// TwinCAT 3 PLC project DAS_CoreSys
// ProgramVersion: 3.1.4024.0
// libraries:
//   AxisInterface_Type03, * (Beckhoff Automation)
//   BATW_Base, * (Beckhoff Automation)
//   Common Behaviour Model, * (3S - Smart Software Solutions GmbH)
//   Tc2_EtherCAT, * (Beckhoff Automation GmbH)
//   Tc2_Math, * (Beckhoff Automation GmbH)
//   Tc2_ModbusRTU, * (Beckhoff Automation GmbH)
//   Tc2_SerialCom, * (Beckhoff Automation GmbH)
//   Tc2_Standard, * (Beckhoff Automation GmbH)
//   Tc2_System, * (Beckhoff Automation GmbH)
//   Tc2_Utilities, * (Beckhoff Automation GmbH)
//   Tc3_JsonXml, * (Beckhoff Automation GmbH)
//   Tc3_MC2_AdvancedHoming, * (Beckhoff Automation GmbH)
//   Tc3_Module, * (Beckhoff Automation GmbH)
//   Tc3_PackML_V2, * (Beckhoff Automation GmbH)
//   Util, * (System)
// project tree:
//   / CoreSys.TcTTO, ModbusTask.TcTTO, MotionSync.TcTTO
//   Library/00_PackML/01_ObjectBase/ eModeChangeState.TcDUT, FB_ModeBase_V1.TcPOU, FB_ModeBase_V2.TcPOU, I_ErrorElement.TcIO, I_ErrorSubject.TcIO
//   Library/00_PackML/02_Mode/ E_Severity.TcDUT, E_UnitMode.TcDUT
//   Library/10_Machine/11_IOData/ GVL_EIP.TcGVL, GVL_Input.TcGVL, GVL_Output.TcGVL
//   Library/10_Machine/12_MachineControl/DUTs/ AxisNo.TcDUT, E_DataFrom.TcDUT, ST_ChangeIntoProduction.TcDUT, ST_CylinderMonitor.TcDUT, ST_MotorMonitor.TcDUT, ST_TableMoveCtrl.TcDUT, ST_TableMoveService.TcDUT, ST_TableMoveStatus.TcDUT, UnitNo.TcDUT
//   Library/10_Machine/12_MachineControl/DUTs/Cylinders/ ST_CylinderList.TcDUT, UNI_CylinderList.TcDUT
//   Library/10_Machine/12_MachineControl/DUTs/FanucRobot/ ST_FanucRobotList.TcDUT, UNI_FanucRobotList.TcDUT
//   Library/10_Machine/12_MachineControl/DUTs/Motor/ ST_MotorList.TcDUT, UNI_MotorList.TcDUT
//   Library/10_Machine/12_MachineControl/DUTs/Service/ ST_ServiceCtrl_Base.TcDUT, ST_ServiceStatus_Base.TcDUT
//   Library/10_Machine/12_MachineControl/DUTs/Setup/ E_ClipNo.TcDUT, ST_AllocateRobotCoordinate.TcDUT, ST_AllocateRobotPositionTable.TcDUT, ST_AxisPara.TcDUT, ST_AxisPara_Auto.TcDUT, ST_AxisPara_HalfAuto.TcDUT, ST_AxisPara_Homing.TcDUT, ST_AxisPara_Manual.TcDUT, ST_CylinderPara.TcDUT, ST_FanucRobotCCDSetting.TcDUT, ST_OutRobotCoordinate.TcDUT, ST_OutRobotPositionTable.TcDUT, ST_PositionTable.TcDUT, ST_SetupAxis.TcDUT, ST_SetupCylinder.TcDUT, ST_SetupFanucRobot.TcDUT, ST_SetupMotor.TcDUT, ST_SetupPara.TcDUT, ST_Setup_Light.TcDUT, ST_Setup_Mechanical.TcDUT
//   Library/10_Machine/12_MachineControl/ FB_MachineControl.TcPOU, GVL_Machine.TcGVL, GVL_Machine_Const.TcGVL
//   Library/10_Machine/12_MachineControl/Service/ FB_MachineHoming.TcPOU
//   Library/10_Machine/18_HMI_Handshake/DUTs/Allocated/ ST_Auto_Allocated.TcDUT, ST_AXIS_HOMING.TcDUT, ST_AXIS_JOG.TcDUT, ST_AXIS_PTP.TcDUT, ST_HalfAuto_Allocated.TcDUT, ST_HMI_ControlOutPut.TcDUT, ST_Manual_Allocated.TcDUT, ST_Manual_NeedleRobot.TcDUT, ST_Manual_Axis.TcDUT, ST_Manual_OutRobot.TcDUT, ST_Manual_PullOutCV.TcDUT, ST_Manual_Allocate.TcDUT, ST_Manual_TransCV.TcDUT, ST_Manual_TurnTable.TcDUT
//   Library/10_Machine/18_HMI_Handshake/DUTs/Component/ ST_DoubleValve.TcDUT, ST_MotorCommand.TcDUT, ST_SignleValve.TcDUT
//   Library/10_Machine/18_HMI_Handshake/DUTs/ E_AllocationJob.TcDUT
//   Library/10_Machine/18_HMI_Handshake/DUTs/IOMonitor/ ST_HMI_ControlInPut.TcDUT, ST_InputTables.TcDUT, ST_Input_IOMonitor.TcDUT, ST_Output_IOMonitor.TcDUT, ST_WheelhouseInput.TcDUT, ST_WheelhouseTour.TcDUT, ST_Wheelhouse_Layer.TcDUT, UNI_HMI_WheelHouseInput.TcDUT, UNI_HMI_WheelHouseInput2.TcDUT (excluded from build)
//   Library/10_Machine/18_HMI_Handshake/DUTs/Shipping/ ST_Auto_Shipping.TcDUT, ST_HalfAuto_Shipping.TcDUT, ST_HMI_ShippingArea.TcDUT, ST_Manual_Shipping.TcDUT
//   Library/10_Machine/18_HMI_Handshake/DUTs/Status/ ST_AllocateStatus.TcDUT, ST_Auto_Status.TcDUT, ST_AXES_STATUS.TcDUT, ST_MotorStatus.TcDUT, ST_SINGLEAXIS_STATUS.TcDUT, ST_CylinderStatus.TcDUT, ST_HalfAuto_Status.TcDUT, ST_HMI_MachineStatus.TcDUT, ST_Manual_Status.TcDUT, ST_ShippingStatus.TcDUT, ST_StorageStatus.TcDUT
//   Library/10_Machine/18_HMI_Handshake/DUTs/Storage/ ST_Auto_Storage.TcDUT, ST_HalfAuto_Storage.TcDUT, ST_HMI_ControlConvery.TcDUT, ST_Manual_FanucRobot.TcDUT, ST_Manual_Rack.TcDUT, ST_Manual_UpCV.TcDUT, ST_Manual_LowCV.TcDUT, ST_Manual_Storage.TcDUT
//   Library/10_Machine/18_HMI_Handshake/ FB_HmiHandShake.TcPOU, GVL_ADS.TcGVL, GVL_HMI.TcGVL
//   Library/10_Machine/18_HMI_Handshake/OLD_DUTs/DataCore/ E_BoxHookPoint.TcDUT, E_BufferArea.TcDUT, E_BoxStatus.TcDUT, E_LayerPoint.TcDUT, E_MachineMode.TcDUT, E_mode.TcDUT, E_NeedleClip.TcDUT, E_Location.TcDUT, E_MachineTask.TcDUT, E_NeedlePoint.TcDUT, E_OutRobotClip.TcDUT, E_OutRobotPoint.TcDUT, E_PlateHookPoint.TcDUT, st_AllocatingNeedleInfo.TcDUT, ST_AllocationJobBatchModeInfo.TcDUT, st_BoxHookStationMove.TcDUT, ST9_ChangeBox.TcDUT, st_ChangeBoxesData.TcDUT, ST0_ChangeBoxesInfo.TcDUT, ST1_ChangeBoxInfo.TcDUT, st_LayerStationMove.TcDUT, ST_Mode.TcDUT, ST_Output.TcDUT, ST_DischargeDataInfo.TcDUT, ST_Feeding.TcDUT, ST_FeedingDataFeeback.TcDUT, ST_FeedingDataInfo.TcDUT, ST_GetBox.TcDUT, st_NeedleAction.TcDUT, st_NeedleActionBatch.TcDUT, ST_NeedleAllocatefeeback.TcDUT, ST_NeedleAllocateinfo.TcDUT, ST_ChangeAllocate.TcDUT, ST_NeedleChangeAllocateInfo.TcDUT, ST_NeedleRemove.TcDUT, ST_NeedleRemoveAllocate.TcDUT, st_OutRobotMove.TcDUT, ST_PCTask.TcDUT, st_PlateHookStationMove.TcDUT, ST_PlateOrder.TcDUT, E_StationOrder.TcDUT, ST_ACTIVEDATA.TcDUT, ST_ActiveResult.TcDUT, ST_AllocationData.TcDUT, ST_AllocationInfo.TcDUT, ST_AllocationJobBatchMode_Reverse.TcDUT, st_ADSBaseParaCore.TcDUT, st_ADSMotoCore.TcDUT, st_ADSMotoMoveCore.TcDUT, st_AllocateParameterCore.TcDUT, st_RegionHome.TcDUT, ST_SheepingPicture.TcDUT, ST_SheepingPictureFeeback.TcDUT, ST_SheepingPictureInfo.TcDUT, ST_SixRobotAction.TcDUT, ST_SixRobotActionFeeback.TcDUT, ST_SixRobotActionInfo.TcDUT, st_SixRobotAreaMove.TcDUT, st_SixRobotPTP.TcDUT, ST_WarehouseBack.TcDUT, ST_WarehouseBackFeeback.TcDUT, ST_WarehouseBackInfo.TcDUT, ST_WarehouseGetBox.TcDUT, ST_ClampingToPlate.TcDUT, st_DASCalibrationData.TcDUT, ST_GetBoxData.TcDUT, ST_GetBoxInfo.TcDUT, ST_InformationExchange.TcDUT, ST_MachineAdjust.TcDUT, ST_MachineTask.TcDUT, ST_Needle.TcDUT, ST_NeedleChageBox.TcDUT, st_NeedleChageBoxData.TcDUT, ST_NeedleWarehouse.TcDUT, ST_NeedleWarehouseData.TcDUT, ST_SixRobotGetOrPut.TcDUT, st_WarehouseData.TcDUT
//   Library/10_Machine/18_HMI_Handshake/Service/DUTs/AllocateBatchMode/ st_AllocateMoveAutoBatchMode_Ctrl.TcDUT, st_AllocateMoveAutoBatchMode_Status.TcDUT, st_Coordinate.TcDUT, ST_Cylinders.TcDUT, st_RoundBeltAutoSingleMove_Ctrl.TcDUT, U_Cylinders.TcDUT
//   Library/10_Machine/18_HMI_Handshake/Service/DUTs/ ST_HMI_Handshake.TcDUT
//   Library/10_Machine/19_Device/EL1889/ ST_EbusDI16.TcDUT, ST_EbusInputModule.TcDUT, ST_InputTable.TcDUT, ST_InputTable_Mitsubishi.TcDUT, uni_InputModule.TcDUT
//   Library/10_Machine/19_Device/EL2889/ ST_EbusDO16.TcDUT, ST_EbusOutputModule.TcDUT, ST_OutputTable.TcDUT, ST_OutputTables.TcDUT, uni_OutputModule.TcDUT
//   Library/10_Machine/19_Device/FanucRobot/DUTs/ E_ClampAction.TcDUT, E_FanucRobotOpMode.TcDUT, E_PullOutConveyorPosition.TcDUT, E_RobotAddress.TcDUT, ST_AutoMode_ShippingRobot_MoveAbs.TcDUT, ST_CCD_ZoneUse.TcDUT, ST_FanucUI1.TcDUT, ST_FanucUO1.TcDUT, ST_Fanuc_AbsMove.TcDUT, ST_Fanuc_GeneralCommand.TcDUT, ST_Fanuc_GeneralCommand_1.TcDUT, ST_Fanuc_Status.TcDUT, ST_Fanuc_WarehouseHandshake.TcDUT, ST_IntToBool.TcDUT, ST_ReadWriteParaCmd.TcDUT, ST_ReadWriteParaStatus.TcDUT
//   Library/10_Machine/19_Device/FanucRobot/ FB_FanucRobot_Basic.TcPOU
//   Library/20_MachineUnits/21_StorageArea/210_Cabinet/DUTs/ E_CabinetJob.TcDUT, st_LayerStatus.TcDUT, st_WarehouseLayer.TcDUT, st_WarehouseList.TcDUT, U_Bits_To_stStatus.TcDUT, _st_LayerStatus.TcDUT, _st_WareHouseLayer.TcDUT, _st_WarehouseList.TcDUT
//   Library/20_MachineUnits/21_StorageArea/210_Cabinet/ FB_WareHouse.TcPOU
//   Library/20_MachineUnits/21_StorageArea/210_Cabinet/Services/ FB_FeedInBox.TcPOU, FB_ReloadBox.TcPOU
//   Library/20_MachineUnits/21_StorageArea/Duts/ E_CabinetJob.TcDUT (excluded from build), E_FeedInAction.TcDUT, E_ReloadRoundBoxAction.TcDUT, st_RobotAbsMove_Ctrl.TcDUT, st_RobotAbsMove_Status.TcDUT, st_RobotWarehouseMove_Ctrl.TcDUT, st_RobotWarehouseMove_Status.TcDUT, ST_StorageService.TcDUT
//   Library/20_MachineUnits/21_StorageArea/ FB_StorageArea.TcPOU
//   Library/20_MachineUnits/21_StorageArea/Service/ FB_AddBoxes_v2.TcPOU, FB_BoxSupplyCtrl.TcPOU, FB_DiameterMovement.TcPOU, FB_FeedInEmptyBoxWithRobot.TcPOU, FB_LowerFeedInConveyor.TcPOU, FB_ReloadRoundBeltBoxWithRobot.TcPOU, FB_RobotAbsMove.TcPOU, FB_RobotRegionMove_AllocatedConveyor.TcPOU, FB_RobotRegionMove_BufferArea.TcPOU, FB_RobotRegionMove_FeedInConveyor.TcPOU, FB_RobotRegionMove_PullOutConveyor.TcPOU, FB_RobotRegionMove_RoundBelt.TcPOU, FB_StorageHoming.TcPOU, FB_UpperFeedInConveyor.TcPOU, FB_WareHouseWithRobotMove.TcPOU
//   Library/20_MachineUnits/22_AllocateArea/Duts/Enums/ E_RoundBeltControlAccess.TcDUT
//   Library/20_MachineUnits/22_AllocateArea/Duts/ E_Pistons.TcDUT, F_Even.TcPOU, ST_AllocateService.TcDUT, ST_DuoCylinders.TcDUT, st_RoundBeltAutoSingleMove_Status.TcDUT, Uni_DuoCylinders.TcDUT
//   Library/20_MachineUnits/22_AllocateArea/ FB_AllocateAreaWithRoundbelt.TcPOU, FB_AllocateAreaWithXPlanar.TcPOU
//   Library/20_MachineUnits/22_AllocateArea/FUNs/ FUN_GetNeedleCoordinates.TcPOU, FUN_GetSyncGroup_AllocationJob.TcPOU
//   Library/20_MachineUnits/22_AllocateArea/Service/ FB_AllocateRobotNeedlingMove.TcPOU, FB_AllocateMoveAutoBatchMode.TcPOU, FB_AllocateMoveAutoBatchMode_Reverse.TcPOU, FB_OutRobot_EmptyBoxMove.TcPOU, FB_OutRobot_RareBoxMove.TcPOU, FB_OutRobot_BoxMoveReverse.TcPOU, FB_OutRobot_BoxMoveTurnTableToRoundBelt.TcPOU, FB_PullOutConveyorAction.TcPOU, FB_PullOutConveyorBtnCtrl.TcPOU, FB_RoundBeltService.TcPOU, FB_AllocateAreaHome.TcPOU, FB_SameSizeCVCamera.TcPOU, FB_DifferentCVCamera.TcPOU, FB_TurnTableService.TcPOU
//   Library/20_MachineUnits/23_ShippingArea/Duts/ ST_ShippingService.TcDUT
//   Library/20_MachineUnits/23_ShippingArea/ FB_ShippingArea.TcPOU
//   Library/20_MachineUnits/23_ShippingArea/Service/ FB_ShippingHoming.TcPOU, FB_ShippingRobot_TransmitCVEnd.TcPOU, FB_ShippingRobot_Left.TcPOU, FB_ShippingRobot_Right.TcPOU
//   Library/99_Utilities/Duts/ E_SignalTowerLampMode.TcDUT, ST_BoolList.TcDUT, ST_SignalTower.TcDUT, uni_IntToBool.TcDUT
//   Library/99_Utilities/ErrorHandling/ FB_ErrorHandler.TcPOU, FB_ErrorHandler_OLD.TcPOU (excluded from build), FB_ErrorHandler_abond.TcPOU (excluded from build), FB_ErrorHandling.TcPOU (excluded from build)
//   Library/99_Utilities/ FB_CylinderManualCtrl.TcPOU, FB_EdgeDetect.TcPOU, FB_MotorManualCtrl.TcPOU, FB_SignalGen.TcPOU, FB_SignalTower.TcPOU, FB_TableMove.TcPOU, FB_XY_Move.TcPOU, FB_XY_PickAndPlace.TcPOU, F_FtoPT.TcPOU
//   Library/99_Utilities/FUNCTION/ FUN_CheckAxisAllowMove.TcPOU, FUN_GetPositionTableData.TcPOU, FUN_MachineState.TcPOU, FUN_ResetStorageCylinder.TcPOU, FUN_RetractStorageCylinder.TcPOU
//   POUs/CheckProg/ CheckBounds.TcPOU, CheckDivDInt.TcPOU, CheckDivLInt.TcPOU, CheckDivLReal.TcPOU, CheckDivReal.TcPOU, CheckLRangeSigned.TcPOU, CheckLRangeUnsigned.TcPOU, CheckPointer.TcPOU, CheckRangeSigned.TcPOU, CheckRangeUnsigned.TcPOU
//   POUs/ DAS_CoreSys.TcPOU, DAS_MotionSync.TcPOU
//   POUs/ModbusRTU/00_BaseFBs/01_FB_ObjectBase/DUTs/ E_MethodStatus_Basic.TcDUT, ST_CmdContent.TcDUT, ST_MsgContent.TcDUT
//   POUs/ModbusRTU/00_BaseFBs/01_FB_ObjectBase/ FB_ObjectBase.TcPOU, FB_ObjectBase_V2.TcPOU
//   POUs/ModbusRTU/00_BaseFBs/01_FB_ObjectBase/GVLs/ Para_ObjectBase.TcGVL
//   POUs/ModbusRTU/00_BaseFBs/01_FB_ObjectBase/ITFs/ IBasicElement.TcIO
//   POUs/ModbusRTU/ ComModbusRTU.TcPOU
//   POUs/ModbusRTU/SerialComTask/DUTs/ un_RS485States.TcDUT, un_RS485States_all.TcDUT
//   POUs/ModbusRTU/SerialComTask/ FB_CommunicateModbusRTU.TcPOU
// real-time tasks:
//   TASK CoreSys: cycle T#10ms, priority 20, ADS port 350
//   TASK MotionSync: cycle T#2ms, priority 1, ADS port 351
//   TASK EIP_Task: cycle T#2ms, priority 2, ADS port 301
//   TASK ModbusTask: cycle T#5ms, priority 21, ADS port 352
// motion (NC):
//   TASK NC-Task 1 SAF: cycle T#2ms, priority 4, ADS port 501
//   TASK NC-Task 1 SVB: cycle T#2ms, priority 8, ADS port 511
//   AXIS Axis 1|TurnTable (id 1)
//     General: UnitName=°
//     Dynamic: Acceleration=1800, Deceleration=1800, Jerk=10800
//     Velo: SlowManual=6, FastManual=60, Maximum=600
//     OtherSettings: AllowMotionCmdToSlave=true
//     encoder EncType=19
//       EncPara: ScaleFactorNumerator=120, ScaleFactorDenominator=83886080, MaxCount=#xffffffff
//         SoftEndMaxControl: Range=350
//         Inc: RefSoftSyncMask=#x0000ffff
//     drive DrvType=16
//       DrvPara: MaxCount=#xffffffff, DriveControlDWord=#x00020100
//         Analog: VeloReferenz=600, TorqueSetpointScale=10, ScaleFactorActTorque=0.1
//         TimeComp: TaskDelayCycles=1
//     controller CtrType=1
//       CtrPara: PriorControlFactor=1
//         PosDiffControl: Enable=false
//         Observer: BandWidth=20
//   AXIS Axis 2|RoundBelt (id 2)
//     General: UnitFlags=#x00000004
//     Dynamic: AccelerationMaximum=3900, DecelerationMaximum=3900, Acceleration=3900, Deceleration=3900, Jerk=30000
//     Velo: SlowManual=6, FastManual=300, Maximum=500
//     OtherSettings: AllowMotionCmdToSlave=true
//     encoder EncType=19
//       EncPara: ScaleFactorNumerator=500, ScaleFactorDenominator=167772160, ModuloFactor=2800, MaxCount=#xffffffff
//         Inc: RefSoftSyncMask=#x0000ffff
//     drive DrvType=16
//       DrvPara: MaxCount=#xffffffff, DriveControlDWord=#x00020100
//         Analog: VeloReferenz=500, TorqueSetpointScale=10, ScaleFactorActTorque=0.1
//         TimeComp: TaskDelayCycles=1
//     controller CtrType=1
//       CtrPara: PriorControlFactor=1
//         PosDiffControl: Range=10
//         Observer: BandWidth=20
//   AXIS Axis 3|AllocateRobot_X (id 3)
//     Dynamic: Acceleration=12000, Deceleration=12000, Jerk=360000
//     Velo: SlowManual=6, FastManual=60, Maximum=800
//     OtherSettings: AllowMotionCmdToSlave=true
//     encoder EncType=19
//       EncPara: ScaleFactorNumerator=36, ScaleFactorDenominator=8388608, MaxCount=#xffffffff
//         Inc: RefSoftSyncMask=#x0000ffff
//     drive DrvType=16
//       DrvPara: MaxCount=#xffffffff, DriveControlDWord=#x00020100
//         Analog: TorqueSetpointScale=10, ScaleFactorActTorque=0.1
//         TimeComp: TaskDelayCycles=1
//     controller CtrType=1
//       CtrPara: PriorControlFactor=1
//         Observer: BandWidth=20
//   AXIS Axis 4|AllocateRobot_Y (id 4)
//     Dynamic: Acceleration=15000, Deceleration=15000, Jerk=225000
//     OtherSettings: AllowMotionCmdToSlave=true
//     encoder EncType=19
//       EncPara: ScaleFactorNumerator=16, ScaleFactorDenominator=8388608, Inverse=true, MaxCount=#xffffffff
//         Inc: RefSoftSyncMask=#x0000ffff
//     drive DrvType=16
//       DrvPara: Inverse=true, MaxCount=#xffffffff, DriveControlDWord=#x00020100
//         Analog: TorqueSetpointScale=10, ScaleFactorActTorque=0.1
//         TimeComp: TaskDelayCycles=1
//     controller CtrType=1
//       CtrPara: PriorControlFactor=1
//         PosDiffControl: Range=10
//         Observer: BandWidth=20
//   AXIS Axis 5|OutRobot_X (id 5)
//     Dynamic: Acceleration=11250, Deceleration=11250, Jerk=168750
//     Velo: SlowManual=6, FastManual=60, Maximum=1500
//     OtherSettings: AllowMotionCmdToSlave=true
//     encoder EncType=19
//       EncPara: ScaleFactorNumerator=30, ScaleFactorDenominator=8388608, MaxCount=#xffffffff
//     drive DrvType=16
//       DrvPara: MaxCount=#xffffffff, DriveControlDWord=#x00020100
//         Analog: TorqueSetpointScale=10, ScaleFactorActTorque=0.1
//         TimeComp: TaskDelayCycles=1
//     controller CtrType=1
//       CtrPara: PriorControlFactor=1
//         PosDiffControl: Range=10
//         Observer: BandWidth=20
//   AXIS Axis 6|OutRobot_Y (id 6)
//     Dynamic: Acceleration=6000, Deceleration=6000, Jerk=36000
//     Velo: SlowManual=6, FastManual=60
//     OtherSettings: AllowMotionCmdToSlave=true
//     encoder EncType=19
//       EncPara: ScaleFactorNumerator=40, ScaleFactorDenominator=8388608, MaxCount=#xffffffff
//     drive DrvType=16
//       DrvPara: MaxCount=#xffffffff, DriveControlDWord=#x00020100
//         Analog: TorqueSetpointScale=10, ScaleFactorActTorque=0.1
//         TimeComp: TaskDelayCycles=1
//     controller CtrType=1
//       CtrPara: PriorControlFactor=1
//         PosDiffControl: Range=10
//         Observer: BandWidth=20
//   AXIS Axis 7|RackMotor (id 7)
//     Dynamic: Acceleration=800.624, Deceleration=800.624, Jerk=1167.58
//     Velo: SlowManual=5, FastManual=100, Maximum=732
//     OtherSettings: AllowMotionCmdToSlave=true
//     encoder EncType=4
//       EncPara: ScaleFactorNumerator=90, ScaleFactorDenominator=980, MaxCount=#xffffffff
//     drive DrvType=23
//       Analog: VeloReferenz=732, TorqueSetpointScale=10, ScaleFactorActTorque=0.1
//       TimeComp: TaskDelayCycles=1
//     controller CtrType=1
//       CtrPara: PriorControlFactor=1
//         PosDiffControl: Enable=false
//         PID: PosKp=90
//         Observer: BandWidth=20
// I/O:
//   DEVICE Device 1 (EtherCAT) Storage, AmsNetId 169.254.53.69.2.1
//     Term 1 (EK1200) [EK1200-5000 EtherCAT Power supply (2A E-Bus)]
//       Term 2 (EL6021) [EL6021 Interface (RS422/485)]
//       Term 3 (EL6021) [EL6021 Interface (RS422/485)]
//       Term 4 (EL6021) [EL6021 Interface (RS422/485)]
//       Term 5 (EL6021) [EL6021 Interface (RS422/485)]
//       Term 6 (EL1889)_01(X6) [EL1889 16Ch. Dig. Input 24V, 3ms, negative]
//       Term 7 (EL1889)_02(X7) [EL1889 16Ch. Dig. Input 24V, 3ms, negative]
//       Term 8 (EL1889)_03(X9) [EL1889 16Ch. Dig. Input 24V, 3ms, negative]
//       Term 9 (EL1889)_04(X10) [EL1889 16Ch. Dig. Input 24V, 3ms, negative]
//       Term 10 (EL2889)_01(Y4) [EL2889 16Ch. Dig. Output 24V, 0.5A, negative]
//       Term 11 (EL2889)_02(Y5) [EL2889 16Ch. Dig. Output 24V, 0.5A, negative]
//       Term 12 (EL2889)_03(Y6) [EL2889 16Ch. Dig. Output 24V, 0.5A, negative]
//       Term 13 (EL2889)_04(Y7) [EL2889 16Ch. Dig. Output 24V, 0.5A, negative]
//       Term 14 (EL2889)_05(Y8) [EL2889 16Ch. Dig. Output 24V, 0.5A, negative]
//       Term 59 (EL9410) [EL9410 E-Bus Power Supplier  (Diagnostics)]
//       Term 15 (EL2889)_06(Y10) [EL2889 16Ch. Dig. Output 24V, 0.5A, negative]
//       Term 17 (EL2889)_07(Y11) [EL2889 16Ch. Dig. Output 24V, 0.5A, negative]
//       Term 18 (EL7342) [EL7342 2Ch. DC motor output stage (50V, 3.5A)]
//       Term 19 (EL6652) [EL6652 EtherNet/IP Scanner (Master)]
//       Term 20 (EL9011) [EL9011 End Terminal]
//   DEVICE Device 4 (EtherCAT) Allocate, AmsNetId 169.254.53.69.5.1
//     Box 21 (CU2508) [CU2508 Ethernet Port]
//     Term 22 (EK1100) [EK1100 EtherCAT Coupler (2A E-Bus)]
//       Term 23 (EL1889)_05(X0) [EL1889 16Ch. Dig. Input 24V, 3ms, negative]
//       Term 24 (EL1889)_06(X1) [EL1889 16Ch. Dig. Input 24V, 3ms, negative]
//       Term 25 (EL1889)_07(X2) [EL1889 16Ch. Dig. Input 24V, 3ms, negative]
//       Term 26 (EL1889)_08(X3) [EL1889 16Ch. Dig. Input 24V, 3ms, negative]
//       Term 27 (EL1889)_09(X8) [EL1889 16Ch. Dig. Input 24V, 3ms, negative]
//       Term 28 (EL1889)_10(X11) [EL1889 16Ch. Dig. Input 24V, 3ms, negative]
//       Term 29 (EL2889)_08(Y0) [EL2889 16Ch. Dig. Output 24V, 0.5A, negative]
//       Term 30 (EL2889)_09(Y1) [EL2889 16Ch. Dig. Output 24V, 0.5A, negative]
//       Term 31 (EL2889)_10(Y2) [EL2889 16Ch. Dig. Output 24V, 0.5A, negative]
//       Term 32 (EL9410) [EL9410 E-Bus Power Supplier  (Diagnostics)]
//       Term 33 (EL1889)_11(X4) [EL1889 16Ch. Dig. Input 24V, 3ms, negative]
//       Term 15 (EL6652) [EL6652 EtherNet/IP Scanner (Master)]
//       Term 16 (EL9011) [EL9011 End Terminal]
//   DEVICE Device 5 (EtherCAT), AmsNetId 169.254.53.69.6.1
//     Box 37 (CU2508) [CU2508 Ethernet Port]
//     Drive 38 (MBDLT25BF) [MBDLT25BF]
//     Drive 39 (MCDLT35BF) [MCDLT35BF]
//     Drive 40 (MBDLT25BF) [MBDLT25BF]
//     Drive 41 (MADLT15BF) [MADLT15BF]
//     Drive 42 (MADLT15BF) [MADLT15BF]
//     Drive 43 (MBDLT25BF) [MBDLT25BF]
//   DEVICE Storage Fanuc Robot (ECAT EIP Scanner (EL6652)), AmsNetId 169.254.53.69.4.1
//     FANUC Robot R30iB+ // <INFO> 192.168.0.3, FANUC Robot R30iB+ (ProdCode: 4, Rev: 3.01, Mac: 00:e0:e4:c5:29:bd) </INFO> <EDS> C:\TwinCAT\3.1\Config\Io\EtherNetIP\FANUCROBOT0301_R30IBP.EDS </EDS>
//   DEVICE Device 6 (ECAT EIP Scanner (EL6652)), AmsNetId 169.254.53.69.7.1
//     FANUC Robot R30iB+ // <INFO> 192.168.0.13, FANUC Robot R30iB+ (ProdCode: 4, Rev: 3.01, Mac: 00:e0:e4:99:c3:31) </INFO> <EDS> C:\TwinCAT\3.1\Config\Io\EtherNetIP\FANUCROBOT0301_R30IBP.EDS </EDS>
//   DEVICE X001 (RT-Ethernet Adapter)
// variable links:
//   NC-Task 1 SAF/Axes/Axis 1|TurnTable <-> Device 5 (EtherCAT)/Drive 38 (MBDLT25BF)
//     Drive/Inputs/In/nDataIn1 <-> Transmit PDO mapping 1/Following error actual value
//     Drive/Inputs/In/nDcOutputTime <-> InfoData/DcOutputShift
//     Drive/Inputs/In/nState1 <-> Transmit PDO mapping 1/Statusword
//     Drive/Inputs/In/nState2 <-> Transmit PDO mapping 1/Statusword @bit 8
//     Drive/Inputs/In/nState4 @bit 1 <-> WcState/InputToggle
//     Drive/Inputs/In/nState4 <-> WcState/WcState
//     Drive/Inputs/In/nState5 <-> Transmit PDO mapping 1/Modes of operation display
//     Drive/Outputs/Out/nCtrl1 <-> Receive PDO mapping 1/Controlword
//     Drive/Outputs/Out/nCtrl2 <-> Receive PDO mapping 1/Controlword @bit 8
//     Drive/Outputs/Out/nCtrl5 <-> Receive PDO mapping 1/Modes of operation
//     Drive/Outputs/Out/nDataOut1 <-> Receive PDO mapping 1/Target position
//     Enc/Inputs/In/nDataIn1 <-> Transmit PDO mapping 1/Position actual value
//     Enc/Inputs/In/nDataIn3 <-> Transmit PDO mapping 1/Touch probe pos1 pos value
//     Enc/Inputs/In/nDcInputTime <-> InfoData/DcInputShift
//     Enc/Inputs/In/nState4 @bit 1 <-> WcState/InputToggle
//     Enc/Inputs/In/nState4 <-> WcState/WcState
//     Enc/Inputs/In/nState5 <-> Transmit PDO mapping 1/Touch probe status
//     Enc/Inputs/In/nState6 <-> Transmit PDO mapping 1/Touch probe status @bit 8
//     Enc/Outputs/Out/nCtrl5 <-> Receive PDO mapping 1/Touch probe function
//     Enc/Outputs/Out/nCtrl6 <-> Receive PDO mapping 1/Touch probe function @bit 8
//   NC-Task 1 SAF/Axes/Axis 2|RoundBelt <-> Device 5 (EtherCAT)/Drive 39 (MCDLT35BF)
//     Drive/Inputs/In/nDataIn1 <-> Transmit PDO mapping 1/Following error actual value
//     Drive/Inputs/In/nDataIn3[0] <-> Transmit PDO mapping 1/Torque actual value
//     Drive/Inputs/In/nDcOutputTime <-> InfoData/DcOutputShift
//     Drive/Inputs/In/nState1 <-> Transmit PDO mapping 1/Statusword
//     Drive/Inputs/In/nState2 <-> Transmit PDO mapping 1/Statusword @bit 8
//     Drive/Inputs/In/nState4 @bit 1 <-> WcState/InputToggle
//     Drive/Inputs/In/nState4 <-> WcState/WcState
//     Drive/Inputs/In/nState5 <-> Transmit PDO mapping 1/Modes of operation display
//     Drive/Outputs/Out/nCtrl1 <-> Receive PDO mapping 1/Controlword
//     Drive/Outputs/Out/nCtrl2 <-> Receive PDO mapping 1/Controlword @bit 8
//     Drive/Outputs/Out/nCtrl5 <-> Receive PDO mapping 1/Modes of operation
//     Drive/Outputs/Out/nDataOut1 <-> Receive PDO mapping 1/Target position
//     Enc/Inputs/In/nDataIn1 <-> Transmit PDO mapping 1/Position actual value
//     Enc/Inputs/In/nDataIn3 <-> Transmit PDO mapping 1/Touch probe pos1 pos value
//     Enc/Inputs/In/nDcInputTime <-> InfoData/DcInputShift
//     Enc/Inputs/In/nState4 @bit 1 <-> WcState/InputToggle
//     Enc/Inputs/In/nState4 <-> WcState/WcState
//     Enc/Inputs/In/nState5 <-> Transmit PDO mapping 1/Touch probe status
//     Enc/Inputs/In/nState6 <-> Transmit PDO mapping 1/Touch probe status @bit 8
//     Enc/Outputs/Out/nCtrl5 <-> Receive PDO mapping 1/Touch probe function
//     Enc/Outputs/Out/nCtrl6 <-> Receive PDO mapping 1/Touch probe function @bit 8
//   NC-Task 1 SAF/Axes/Axis 3|AllocateRobot_X <-> Device 5 (EtherCAT)/Drive 40 (MBDLT25BF)
//     Drive/Inputs/In/nDataIn1 <-> Transmit PDO mapping 1/Following error actual value
//     Drive/Inputs/In/nDcOutputTime <-> InfoData/DcOutputShift
//     Drive/Inputs/In/nState1 <-> Transmit PDO mapping 1/Statusword
//     Drive/Inputs/In/nState2 <-> Transmit PDO mapping 1/Statusword @bit 8
//     Drive/Inputs/In/nState4 @bit 1 <-> WcState/InputToggle
//     Drive/Inputs/In/nState4 <-> WcState/WcState
//     Drive/Inputs/In/nState5 <-> Transmit PDO mapping 1/Modes of operation display
//     Drive/Outputs/Out/nCtrl1 <-> Receive PDO mapping 1/Controlword
//     Drive/Outputs/Out/nCtrl2 <-> Receive PDO mapping 1/Controlword @bit 8
//     Drive/Outputs/Out/nCtrl5 <-> Receive PDO mapping 1/Modes of operation
//     Drive/Outputs/Out/nDataOut1 <-> Receive PDO mapping 1/Target position
//     Enc/Inputs/In/nDataIn1 <-> Transmit PDO mapping 1/Position actual value
//     Enc/Inputs/In/nDataIn3 <-> Transmit PDO mapping 1/Touch probe pos1 pos value
//     Enc/Inputs/In/nDcInputTime <-> InfoData/DcInputShift
//     Enc/Inputs/In/nState4 @bit 1 <-> WcState/InputToggle
//     Enc/Inputs/In/nState4 <-> WcState/WcState
//     Enc/Inputs/In/nState5 <-> Transmit PDO mapping 1/Touch probe status
//     Enc/Inputs/In/nState6 <-> Transmit PDO mapping 1/Touch probe status @bit 8
//     Enc/Outputs/Out/nCtrl5 <-> Receive PDO mapping 1/Touch probe function
//     Enc/Outputs/Out/nCtrl6 <-> Receive PDO mapping 1/Touch probe function @bit 8
//   NC-Task 1 SAF/Axes/Axis 4|AllocateRobot_Y <-> Device 5 (EtherCAT)/Drive 41 (MADLT15BF)
//     Drive/Inputs/In/nDataIn1 <-> Transmit PDO mapping 1/Following error actual value
//     Drive/Inputs/In/nDcOutputTime <-> InfoData/DcOutputShift
//     Drive/Inputs/In/nState1 <-> Transmit PDO mapping 1/Statusword
//     Drive/Inputs/In/nState2 <-> Transmit PDO mapping 1/Statusword @bit 8
//     Drive/Inputs/In/nState4 @bit 1 <-> WcState/InputToggle
//     Drive/Inputs/In/nState4 <-> WcState/WcState
//     Drive/Inputs/In/nState5 <-> Transmit PDO mapping 1/Modes of operation display
//     Drive/Outputs/Out/nCtrl1 <-> Receive PDO mapping 1/Controlword
//     Drive/Outputs/Out/nCtrl2 <-> Receive PDO mapping 1/Controlword @bit 8
//     Drive/Outputs/Out/nCtrl5 <-> Receive PDO mapping 1/Modes of operation
//     Drive/Outputs/Out/nDataOut1 <-> Receive PDO mapping 1/Target position
//     Enc/Inputs/In/nDataIn1 <-> Transmit PDO mapping 1/Position actual value
//     Enc/Inputs/In/nDataIn3 <-> Transmit PDO mapping 1/Touch probe pos1 pos value
//     Enc/Inputs/In/nDcInputTime <-> InfoData/DcInputShift
//     Enc/Inputs/In/nState4 @bit 1 <-> WcState/InputToggle
//     Enc/Inputs/In/nState4 <-> WcState/WcState
//     Enc/Inputs/In/nState5 <-> Transmit PDO mapping 1/Touch probe status
//     Enc/Inputs/In/nState6 <-> Transmit PDO mapping 1/Touch probe status @bit 8
//     Enc/Outputs/Out/nCtrl5 <-> Receive PDO mapping 1/Touch probe function
//     Enc/Outputs/Out/nCtrl6 <-> Receive PDO mapping 1/Touch probe function @bit 8
//   NC-Task 1 SAF/Axes/Axis 5|OutRobot_X <-> Device 5 (EtherCAT)/Drive 42 (MADLT15BF)
//     Drive/Inputs/In/nDataIn1 <-> Transmit PDO mapping 1/Following error actual value
//     Drive/Inputs/In/nDcOutputTime <-> InfoData/DcOutputShift
//     Drive/Inputs/In/nState1 <-> Transmit PDO mapping 1/Statusword
//     Drive/Inputs/In/nState2 <-> Transmit PDO mapping 1/Statusword @bit 8
//     Drive/Inputs/In/nState4 @bit 1 <-> WcState/InputToggle
//     Drive/Inputs/In/nState4 <-> WcState/WcState
//     Drive/Inputs/In/nState5 <-> Transmit PDO mapping 1/Modes of operation display
//     Drive/Outputs/Out/nCtrl1 <-> Receive PDO mapping 1/Controlword
//     Drive/Outputs/Out/nCtrl2 <-> Receive PDO mapping 1/Controlword @bit 8
//     Drive/Outputs/Out/nCtrl5 <-> Receive PDO mapping 1/Modes of operation
//     Drive/Outputs/Out/nDataOut1 <-> Receive PDO mapping 1/Target position
//     Enc/Inputs/In/nDataIn1 <-> Transmit PDO mapping 1/Position actual value
//     Enc/Inputs/In/nDataIn3 <-> Transmit PDO mapping 1/Touch probe pos1 pos value
//     Enc/Inputs/In/nDcInputTime <-> InfoData/DcInputShift
//     Enc/Inputs/In/nState4 @bit 1 <-> WcState/InputToggle
//     Enc/Inputs/In/nState4 <-> WcState/WcState
//     Enc/Inputs/In/nState5 <-> Transmit PDO mapping 1/Touch probe status
//     Enc/Inputs/In/nState6 <-> Transmit PDO mapping 1/Touch probe status @bit 8
//     Enc/Outputs/Out/nCtrl5 <-> Receive PDO mapping 1/Touch probe function
//     Enc/Outputs/Out/nCtrl6 <-> Receive PDO mapping 1/Touch probe function @bit 8
//   NC-Task 1 SAF/Axes/Axis 6|OutRobot_Y <-> Device 5 (EtherCAT)/Drive 43 (MBDLT25BF)
//     Drive/Inputs/In/nDataIn1 <-> Transmit PDO mapping 1/Following error actual value
//     Drive/Inputs/In/nDcOutputTime <-> InfoData/DcOutputShift
//     Drive/Inputs/In/nState1 <-> Transmit PDO mapping 1/Statusword
//     Drive/Inputs/In/nState2 <-> Transmit PDO mapping 1/Statusword @bit 8
//     Drive/Inputs/In/nState4 @bit 1 <-> WcState/InputToggle
//     Drive/Inputs/In/nState4 <-> WcState/WcState
//     Drive/Inputs/In/nState5 <-> Transmit PDO mapping 1/Modes of operation display
//     Drive/Outputs/Out/nCtrl1 <-> Receive PDO mapping 1/Controlword
//     Drive/Outputs/Out/nCtrl2 <-> Receive PDO mapping 1/Controlword @bit 8
//     Drive/Outputs/Out/nCtrl5 <-> Receive PDO mapping 1/Modes of operation
//     Drive/Outputs/Out/nDataOut1 <-> Receive PDO mapping 1/Target position
//     Enc/Inputs/In/nDataIn1 <-> Transmit PDO mapping 1/Position actual value
//     Enc/Inputs/In/nDataIn3 <-> Transmit PDO mapping 1/Touch probe pos1 pos value
//     Enc/Inputs/In/nDcInputTime <-> InfoData/DcInputShift
//     Enc/Inputs/In/nState4 @bit 1 <-> WcState/InputToggle
//     Enc/Inputs/In/nState4 <-> WcState/WcState
//     Enc/Inputs/In/nState5 <-> Transmit PDO mapping 1/Touch probe status
//     Enc/Inputs/In/nState6 <-> Transmit PDO mapping 1/Touch probe status @bit 8
//     Enc/Outputs/Out/nCtrl5 <-> Receive PDO mapping 1/Touch probe function
//     Enc/Outputs/Out/nCtrl6 <-> Receive PDO mapping 1/Touch probe function @bit 8
//   NC-Task 1 SAF/Axes/Axis 7|RackMotor <-> Device 1 (EtherCAT) Storage/Term 1 (EK1200)/Term 18 (EL7342)
//     Drive/Inputs/In/nState1 @bit 3 <-> DCM Status Channel 1/Status/Error
//     Drive/Inputs/In/nState1 @bit 5 <-> DCM Status Channel 1/Status/Moving negative
//     Drive/Inputs/In/nState1 @bit 4 <-> DCM Status Channel 1/Status/Moving positive
//     Drive/Inputs/In/nState1 @bit 1 <-> DCM Status Channel 1/Status/Ready
//     Drive/Inputs/In/nState1 <-> DCM Status Channel 1/Status/Ready to enable
//     Drive/Inputs/In/nState1 @bit 6 <-> DCM Status Channel 1/Status/Torque reduced
//     Drive/Inputs/In/nState1 @bit 2 <-> DCM Status Channel 1/Status/Warning
//     Drive/Inputs/In/nState2 @bit 3 <-> DCM Status Channel 1/Status/Digital input 1
//     Drive/Inputs/In/nState2 @bit 4 <-> DCM Status Channel 1/Status/Digital input 2
//     Drive/Inputs/In/nState2 @bit 5 <-> DCM Status Channel 1/Status/Sync error
//     Drive/Inputs/In/nState2 @bit 7 <-> DCM Status Channel 1/Status/TxPDO Toggle
//     Drive/Inputs/In/nState4 @bit 1 <-> WcState/InputToggle
//     Drive/Inputs/In/nState4 <-> WcState/WcState
//     Drive/Outputs/Out/nCtrl1 <-> DCM Control Channel 1/Control/Enable
//     Drive/Outputs/Out/nCtrl1 @bit 2 <-> DCM Control Channel 1/Control/Reduce torque
//     Drive/Outputs/Out/nCtrl1 @bit 1 <-> DCM Control Channel 1/Control/Reset
//     Drive/Outputs/Out/nCtrl1 @bit 3 <-> DCM Control Channel 1/Control/Threshold active
//     Drive/Outputs/Out/nDataOut2[0] <-> DCM Velocity Channel 1/Velocity
//     Enc/Inputs/In/nDataIn1 <-> ENC Status Channel 1/Counter value
//     Enc/Inputs/In/nDataIn2 <-> ENC Status Channel 1/Latch value
//     Enc/Inputs/In/nState1 @bit 4 <-> ENC Status Channel 1/Status/Counter overflow
//     Enc/Inputs/In/nState1 @bit 3 <-> ENC Status Channel 1/Status/Counter underflow
//     Enc/Inputs/In/nState1 @bit 7 <-> ENC Status Channel 1/Status/Extrapolation stall
//     Enc/Inputs/In/nState1 @bit 1 <-> ENC Status Channel 1/Status/Latch extern valid
//     Enc/Inputs/In/nState1 @bit 2 <-> ENC Status Channel 1/Status/Set counter done
//     Enc/Inputs/In/nState2 @bit 4 <-> ENC Status Channel 1/Status/Status of extern latch
//     Enc/Inputs/In/nState2 <-> ENC Status Channel 1/Status/Status of input A
//     Enc/Inputs/In/nState2 @bit 1 <-> ENC Status Channel 1/Status/Status of input B
//     Enc/Inputs/In/nState2 @bit 5 <-> ENC Status Channel 1/Status/Sync error
//     Enc/Inputs/In/nState2 @bit 7 <-> ENC Status Channel 1/Status/TxPDO Toggle
//     Enc/Inputs/In/nState4 @bit 1 <-> WcState/InputToggle
//     Enc/Inputs/In/nState4 <-> WcState/WcState
//     Enc/Outputs/Out/nCtrl1 @bit 3 <-> ENC Control Channel 1/Control/Enable latch extern on negative edge
//     Enc/Outputs/Out/nCtrl1 @bit 1 <-> ENC Control Channel 1/Control/Enable latch extern on positive edge
//     Enc/Outputs/Out/nCtrl1 @bit 2 <-> ENC Control Channel 1/Control/Set counter
//     Enc/Outputs/Out/nDataOut1 <-> ENC Control Channel 1/Set counter value
//   DAS_CoreSys/DAS_CoreSys Instance <-> Device 1 (EtherCAT) Storage/Term 1 (EK1200)/Term 10 (EL2889)_01(Y4)
//     ModbusTask Outputs/GVL_Output.uniDO.stEbusDO.EL2889_01.DO1 <-> Channel 1/Output
//     ModbusTask Outputs/GVL_Output.uniDO.stEbusDO.EL2889_01.DO10 <-> Channel 10/Output
//     ModbusTask Outputs/GVL_Output.uniDO.stEbusDO.EL2889_01.DO11 <-> Channel 11/Output
//     ModbusTask Outputs/GVL_Output.uniDO.stEbusDO.EL2889_01.DO12 <-> Channel 12/Output
//     ModbusTask Outputs/GVL_Output.uniDO.stEbusDO.EL2889_01.DO13 <-> Channel 13/Output
//     ModbusTask Outputs/GVL_Output.uniDO.stEbusDO.EL2889_01.DO14 <-> Channel 14/Output
//     ModbusTask Outputs/GVL_Output.uniDO.stEbusDO.EL2889_01.DO15 <-> Channel 15/Output
//     ModbusTask Outputs/GVL_Output.uniDO.stEbusDO.EL2889_01.DO16 <-> Channel 16/Output
//     ModbusTask Outputs/GVL_Output.uniDO.stEbusDO.EL2889_01.DO2 <-> Channel 2/Output
//     ModbusTask Outputs/GVL_Output.uniDO.stEbusDO.EL2889_01.DO3 <-> Channel 3/Output
//     ModbusTask Outputs/GVL_Output.uniDO.stEbusDO.EL2889_01.DO4 <-> Channel 4/Output
//     ModbusTask Outputs/GVL_Output.uniDO.stEbusDO.EL2889_01.DO5 <-> Channel 5/Output
//     ModbusTask Outputs/GVL_Output.uniDO.stEbusDO.EL2889_01.DO6 <-> Channel 6/Output
//     ModbusTask Outputs/GVL_Output.uniDO.stEbusDO.EL2889_01.DO7 <-> Channel 7/Output
//     ModbusTask Outputs/GVL_Output.uniDO.stEbusDO.EL2889_01.DO8 <-> Channel 8/Output
//     ModbusTask Outputs/GVL_Output.uniDO.stEbusDO.EL2889_01.DO9 <-> Channel 9/Output
//   DAS_CoreSys/DAS_CoreSys Instance <-> Device 1 (EtherCAT) Storage/Term 1 (EK1200)/Term 11 (EL2889)_02(Y5)
//     ModbusTask Outputs/GVL_Output.uniDO.stEbusDO.EL2889_02.DO1 <-> Channel 1/Output
//     ModbusTask Outputs/GVL_Output.uniDO.stEbusDO.EL2889_02.DO10 <-> Channel 10/Output
//     ModbusTask Outputs/GVL_Output.uniDO.stEbusDO.EL2889_02.DO11 <-> Channel 11/Output
//     ModbusTask Outputs/GVL_Output.uniDO.stEbusDO.EL2889_02.DO12 <-> Channel 12/Output
//     ModbusTask Outputs/GVL_Output.uniDO.stEbusDO.EL2889_02.DO13 <-> Channel 13/Output
//     ModbusTask Outputs/GVL_Output.uniDO.stEbusDO.EL2889_02.DO14 <-> Channel 14/Output
//     ModbusTask Outputs/GVL_Output.uniDO.stEbusDO.EL2889_02.DO15 <-> Channel 15/Output
//     ModbusTask Outputs/GVL_Output.uniDO.stEbusDO.EL2889_02.DO16 <-> Channel 16/Output
//     ModbusTask Outputs/GVL_Output.uniDO.stEbusDO.EL2889_02.DO2 <-> Channel 2/Output
//     ModbusTask Outputs/GVL_Output.uniDO.stEbusDO.EL2889_02.DO3 <-> Channel 3/Output
//     ModbusTask Outputs/GVL_Output.uniDO.stEbusDO.EL2889_02.DO4 <-> Channel 4/Output
//     ModbusTask Outputs/GVL_Output.uniDO.stEbusDO.EL2889_02.DO5 <-> Channel 5/Output
//     ModbusTask Outputs/GVL_Output.uniDO.stEbusDO.EL2889_02.DO6 <-> Channel 6/Output
//     ModbusTask Outputs/GVL_Output.uniDO.stEbusDO.EL2889_02.DO7 <-> Channel 7/Output
//     ModbusTask Outputs/GVL_Output.uniDO.stEbusDO.EL2889_02.DO8 <-> Channel 8/Output
//     ModbusTask Outputs/GVL_Output.uniDO.stEbusDO.EL2889_02.DO9 <-> Channel 9/Output
//   DAS_CoreSys/DAS_CoreSys Instance <-> Device 1 (EtherCAT) Storage/Term 1 (EK1200)/Term 12 (EL2889)_03(Y6)
//     ModbusTask Outputs/GVL_Output.uniDO.stEbusDO.EL2889_03.DO1 <-> Channel 1/Output
//     ModbusTask Outputs/GVL_Output.uniDO.stEbusDO.EL2889_03.DO10 <-> Channel 10/Output
//     ModbusTask Outputs/GVL_Output.uniDO.stEbusDO.EL2889_03.DO11 <-> Channel 11/Output
//     ModbusTask Outputs/GVL_Output.uniDO.stEbusDO.EL2889_03.DO12 <-> Channel 12/Output
//     ModbusTask Outputs/GVL_Output.uniDO.stEbusDO.EL2889_03.DO13 <-> Channel 13/Output
//     ModbusTask Outputs/GVL_Output.uniDO.stEbusDO.EL2889_03.DO14 <-> Channel 14/Output
//     ModbusTask Outputs/GVL_Output.uniDO.stEbusDO.EL2889_03.DO15 <-> Channel 15/Output
//     ModbusTask Outputs/GVL_Output.uniDO.stEbusDO.EL2889_03.DO16 <-> Channel 16/Output
//     ModbusTask Outputs/GVL_Output.uniDO.stEbusDO.EL2889_03.DO2 <-> Channel 2/Output
//     ModbusTask Outputs/GVL_Output.uniDO.stEbusDO.EL2889_03.DO3 <-> Channel 3/Output
//     ModbusTask Outputs/GVL_Output.uniDO.stEbusDO.EL2889_03.DO4 <-> Channel 4/Output
//     ModbusTask Outputs/GVL_Output.uniDO.stEbusDO.EL2889_03.DO5 <-> Channel 5/Output
//     ModbusTask Outputs/GVL_Output.uniDO.stEbusDO.EL2889_03.DO6 <-> Channel 6/Output
//     ModbusTask Outputs/GVL_Output.uniDO.stEbusDO.EL2889_03.DO7 <-> Channel 7/Output
//     ModbusTask Outputs/GVL_Output.uniDO.stEbusDO.EL2889_03.DO8 <-> Channel 8/Output
//     ModbusTask Outputs/GVL_Output.uniDO.stEbusDO.EL2889_03.DO9 <-> Channel 9/Output
//   DAS_CoreSys/DAS_CoreSys Instance <-> Device 1 (EtherCAT) Storage/Term 1 (EK1200)/Term 13 (EL2889)_04(Y7)
//     ModbusTask Outputs/GVL_Output.uniDO.stEbusDO.EL2889_04.DO1 <-> Channel 1/Output
//     ModbusTask Outputs/GVL_Output.uniDO.stEbusDO.EL2889_04.DO10 <-> Channel 10/Output
//     ModbusTask Outputs/GVL_Output.uniDO.stEbusDO.EL2889_04.DO11 <-> Channel 11/Output
//     ModbusTask Outputs/GVL_Output.uniDO.stEbusDO.EL2889_04.DO12 <-> Channel 12/Output
//     ModbusTask Outputs/GVL_Output.uniDO.stEbusDO.EL2889_04.DO13 <-> Channel 13/Output
//     ModbusTask Outputs/GVL_Output.uniDO.stEbusDO.EL2889_04.DO14 <-> Channel 14/Output
//     ModbusTask Outputs/GVL_Output.uniDO.stEbusDO.EL2889_04.DO15 <-> Channel 15/Output
//     ModbusTask Outputs/GVL_Output.uniDO.stEbusDO.EL2889_04.DO16 <-> Channel 16/Output
//     ModbusTask Outputs/GVL_Output.uniDO.stEbusDO.EL2889_04.DO2 <-> Channel 2/Output
//     ModbusTask Outputs/GVL_Output.uniDO.stEbusDO.EL2889_04.DO3 <-> Channel 3/Output
//     ModbusTask Outputs/GVL_Output.uniDO.stEbusDO.EL2889_04.DO4 <-> Channel 4/Output
//     ModbusTask Outputs/GVL_Output.uniDO.stEbusDO.EL2889_04.DO5 <-> Channel 5/Output
//     ModbusTask Outputs/GVL_Output.uniDO.stEbusDO.EL2889_04.DO6 <-> Channel 6/Output
//     ModbusTask Outputs/GVL_Output.uniDO.stEbusDO.EL2889_04.DO7 <-> Channel 7/Output
//     ModbusTask Outputs/GVL_Output.uniDO.stEbusDO.EL2889_04.DO8 <-> Channel 8/Output
//     ModbusTask Outputs/GVL_Output.uniDO.stEbusDO.EL2889_04.DO9 <-> Channel 9/Output
//   DAS_CoreSys/DAS_CoreSys Instance <-> Device 1 (EtherCAT) Storage/Term 1 (EK1200)/Term 14 (EL2889)_05(Y8)
//     ModbusTask Outputs/GVL_Output.uniDO.stEbusDO.EL2889_05.DO1 <-> Channel 1/Output
//     ModbusTask Outputs/GVL_Output.uniDO.stEbusDO.EL2889_05.DO10 <-> Channel 10/Output
//     ModbusTask Outputs/GVL_Output.uniDO.stEbusDO.EL2889_05.DO11 <-> Channel 11/Output
//     ModbusTask Outputs/GVL_Output.uniDO.stEbusDO.EL2889_05.DO12 <-> Channel 12/Output
//     ModbusTask Outputs/GVL_Output.uniDO.stEbusDO.EL2889_05.DO13 <-> Channel 13/Output
//     ModbusTask Outputs/GVL_Output.uniDO.stEbusDO.EL2889_05.DO14 <-> Channel 14/Output
//     ModbusTask Outputs/GVL_Output.uniDO.stEbusDO.EL2889_05.DO15 <-> Channel 15/Output
//     ModbusTask Outputs/GVL_Output.uniDO.stEbusDO.EL2889_05.DO16 <-> Channel 16/Output
//     ModbusTask Outputs/GVL_Output.uniDO.stEbusDO.EL2889_05.DO2 <-> Channel 2/Output
//     ModbusTask Outputs/GVL_Output.uniDO.stEbusDO.EL2889_05.DO3 <-> Channel 3/Output
//     ModbusTask Outputs/GVL_Output.uniDO.stEbusDO.EL2889_05.DO4 <-> Channel 4/Output
//     ModbusTask Outputs/GVL_Output.uniDO.stEbusDO.EL2889_05.DO5 <-> Channel 5/Output
//     ModbusTask Outputs/GVL_Output.uniDO.stEbusDO.EL2889_05.DO6 <-> Channel 6/Output
//     ModbusTask Outputs/GVL_Output.uniDO.stEbusDO.EL2889_05.DO7 <-> Channel 7/Output
//     ModbusTask Outputs/GVL_Output.uniDO.stEbusDO.EL2889_05.DO8 <-> Channel 8/Output
//     ModbusTask Outputs/GVL_Output.uniDO.stEbusDO.EL2889_05.DO9 <-> Channel 9/Output
//   DAS_CoreSys/DAS_CoreSys Instance <-> Device 1 (EtherCAT) Storage/Term 1 (EK1200)/Term 15 (EL2889)_06(Y10)
//     ModbusTask Outputs/GVL_Output.uniDO.stEbusDO.EL2889_06.DO1 <-> Channel 1/Output
//     ModbusTask Outputs/GVL_Output.uniDO.stEbusDO.EL2889_06.DO10 <-> Channel 10/Output
//     ModbusTask Outputs/GVL_Output.uniDO.stEbusDO.EL2889_06.DO11 <-> Channel 11/Output
//     ModbusTask Outputs/GVL_Output.uniDO.stEbusDO.EL2889_06.DO12 <-> Channel 12/Output
//     ModbusTask Outputs/GVL_Output.uniDO.stEbusDO.EL2889_06.DO13 <-> Channel 13/Output
//     ModbusTask Outputs/GVL_Output.uniDO.stEbusDO.EL2889_06.DO14 <-> Channel 14/Output
//     ModbusTask Outputs/GVL_Output.uniDO.stEbusDO.EL2889_06.DO15 <-> Channel 15/Output
//     ModbusTask Outputs/GVL_Output.uniDO.stEbusDO.EL2889_06.DO16 <-> Channel 16/Output
//     ModbusTask Outputs/GVL_Output.uniDO.stEbusDO.EL2889_06.DO2 <-> Channel 2/Output
//     ModbusTask Outputs/GVL_Output.uniDO.stEbusDO.EL2889_06.DO3 <-> Channel 3/Output
//     ModbusTask Outputs/GVL_Output.uniDO.stEbusDO.EL2889_06.DO4 <-> Channel 4/Output
//     ModbusTask Outputs/GVL_Output.uniDO.stEbusDO.EL2889_06.DO5 <-> Channel 5/Output
//     ModbusTask Outputs/GVL_Output.uniDO.stEbusDO.EL2889_06.DO6 <-> Channel 6/Output
//     ModbusTask Outputs/GVL_Output.uniDO.stEbusDO.EL2889_06.DO7 <-> Channel 7/Output
//     ModbusTask Outputs/GVL_Output.uniDO.stEbusDO.EL2889_06.DO8 <-> Channel 8/Output
//     ModbusTask Outputs/GVL_Output.uniDO.stEbusDO.EL2889_06.DO9 <-> Channel 9/Output
//   DAS_CoreSys/DAS_CoreSys Instance <-> Device 1 (EtherCAT) Storage/Term 1 (EK1200)/Term 17 (EL2889)_07(Y11)
//     ModbusTask Outputs/GVL_Output.uniDO.stEbusDO.EL2889_07.DO1 <-> Channel 1/Output
//     ModbusTask Outputs/GVL_Output.uniDO.stEbusDO.EL2889_07.DO10 <-> Channel 10/Output
//     ModbusTask Outputs/GVL_Output.uniDO.stEbusDO.EL2889_07.DO11 <-> Channel 11/Output
//     ModbusTask Outputs/GVL_Output.uniDO.stEbusDO.EL2889_07.DO12 <-> Channel 12/Output
//     ModbusTask Outputs/GVL_Output.uniDO.stEbusDO.EL2889_07.DO13 <-> Channel 13/Output
//     ModbusTask Outputs/GVL_Output.uniDO.stEbusDO.EL2889_07.DO14 <-> Channel 14/Output
//     ModbusTask Outputs/GVL_Output.uniDO.stEbusDO.EL2889_07.DO15 <-> Channel 15/Output
//     ModbusTask Outputs/GVL_Output.uniDO.stEbusDO.EL2889_07.DO16 <-> Channel 16/Output
//     ModbusTask Outputs/GVL_Output.uniDO.stEbusDO.EL2889_07.DO2 <-> Channel 2/Output
//     ModbusTask Outputs/GVL_Output.uniDO.stEbusDO.EL2889_07.DO3 <-> Channel 3/Output
//     ModbusTask Outputs/GVL_Output.uniDO.stEbusDO.EL2889_07.DO4 <-> Channel 4/Output
//     ModbusTask Outputs/GVL_Output.uniDO.stEbusDO.EL2889_07.DO5 <-> Channel 5/Output
//     ModbusTask Outputs/GVL_Output.uniDO.stEbusDO.EL2889_07.DO6 <-> Channel 6/Output
//     ModbusTask Outputs/GVL_Output.uniDO.stEbusDO.EL2889_07.DO7 <-> Channel 7/Output
//     ModbusTask Outputs/GVL_Output.uniDO.stEbusDO.EL2889_07.DO8 <-> Channel 8/Output
//     ModbusTask Outputs/GVL_Output.uniDO.stEbusDO.EL2889_07.DO9 <-> Channel 9/Output
//   DAS_CoreSys/DAS_CoreSys Instance <-> Device 1 (EtherCAT) Storage/Term 1 (EK1200)/Term 2 (EL6021)
//     CoreSys Inputs/ComModbusRTU.MBdata_Read_ControllerN[3][{0..21}] <-> COM TxPDO-Map Inputs/Data In {0..21}  (22 links)
//     CoreSys Inputs/ComModbusRTU.fb_Warehouse_Modbus[3].MB_EL6X22B_ControllerN.InData/D[{0..21}] <-> COM TxPDO-Map Inputs/Data In {0..21}  (22 links)
//     CoreSys Inputs/ComModbusRTU.fb_Warehouse_Modbus[3].MB_EL6X22B_ControllerN.InData/Status <-> COM TxPDO-Map Inputs/Status
//     CoreSys Outputs/ComModbusRTU.fb_Warehouse_Modbus[3].MB_EL6X22B_ControllerN.OutData/Ctrl <-> COM RxPDO-Map Outputs/Ctrl
//     CoreSys Outputs/ComModbusRTU.fb_Warehouse_Modbus[3].MB_EL6X22B_ControllerN.OutData/D[{0..21}] <-> COM RxPDO-Map Outputs/Data Out {0..21}  (22 links)
//   DAS_CoreSys/DAS_CoreSys Instance <-> Device 1 (EtherCAT) Storage/Term 1 (EK1200)/Term 3 (EL6021)
//     CoreSys Inputs/ComModbusRTU.MBdata_Read_ControllerN[2][{0..21}] <-> COM TxPDO-Map Inputs/Data In {0..21}  (22 links)
//     CoreSys Inputs/ComModbusRTU.fb_Warehouse_Modbus[2].MB_EL6X22B_ControllerN.InData/D[{0..21}] <-> COM TxPDO-Map Inputs/Data In {0..21}  (22 links)
//     CoreSys Inputs/ComModbusRTU.fb_Warehouse_Modbus[2].MB_EL6X22B_ControllerN.InData/Status <-> COM TxPDO-Map Inputs/Status
//     CoreSys Outputs/ComModbusRTU.fb_Warehouse_Modbus[2].MB_EL6X22B_ControllerN.OutData/Ctrl <-> COM RxPDO-Map Outputs/Ctrl
//     CoreSys Outputs/ComModbusRTU.fb_Warehouse_Modbus[2].MB_EL6X22B_ControllerN.OutData/D[{0..21}] <-> COM RxPDO-Map Outputs/Data Out {0..21}  (22 links)
//   DAS_CoreSys/DAS_CoreSys Instance <-> Device 1 (EtherCAT) Storage/Term 1 (EK1200)/Term 4 (EL6021)
//     CoreSys Inputs/ComModbusRTU.MBdata_Read_ControllerN[1][{0..21}] <-> COM TxPDO-Map Inputs/Data In {0..21}  (22 links)
//     CoreSys Inputs/ComModbusRTU.fb_Warehouse_Modbus[1].MB_EL6X22B_ControllerN.InData/D[{0..21}] <-> COM TxPDO-Map Inputs/Data In {0..21}  (22 links)
//     CoreSys Inputs/ComModbusRTU.fb_Warehouse_Modbus[1].MB_EL6X22B_ControllerN.InData/Status <-> COM TxPDO-Map Inputs/Status
//     CoreSys Outputs/ComModbusRTU.fb_Warehouse_Modbus[1].MB_EL6X22B_ControllerN.OutData/Ctrl <-> COM RxPDO-Map Outputs/Ctrl
//     CoreSys Outputs/ComModbusRTU.fb_Warehouse_Modbus[1].MB_EL6X22B_ControllerN.OutData/D[{0..21}] <-> COM RxPDO-Map Outputs/Data Out {0..21}  (22 links)
//   DAS_CoreSys/DAS_CoreSys Instance <-> Device 1 (EtherCAT) Storage/Term 1 (EK1200)/Term 5 (EL6021)
//     CoreSys Inputs/ComModbusRTU.MBdata_Read_ControllerN[0][{0..21}] <-> COM TxPDO-Map Inputs/Data In {0..21}  (22 links)
//     CoreSys Inputs/ComModbusRTU.fb_Warehouse_Modbus[0].MB_EL6X22B_ControllerN.InData/D[{0..21}] <-> COM TxPDO-Map Inputs/Data In {0..21}  (22 links)
//     CoreSys Inputs/ComModbusRTU.fb_Warehouse_Modbus[0].MB_EL6X22B_ControllerN.InData/Status <-> COM TxPDO-Map Inputs/Status
//     CoreSys Outputs/ComModbusRTU.fb_Warehouse_Modbus[0].MB_EL6X22B_ControllerN.OutData/Ctrl <-> COM RxPDO-Map Outputs/Ctrl
//     CoreSys Outputs/ComModbusRTU.fb_Warehouse_Modbus[0].MB_EL6X22B_ControllerN.OutData/D[{0..21}] <-> COM RxPDO-Map Outputs/Data Out {0..21}  (22 links)
//   DAS_CoreSys/DAS_CoreSys Instance <-> Device 1 (EtherCAT) Storage/Term 1 (EK1200)/Term 6 (EL1889)_01(X6)
//     ModbusTask Inputs/GVL_Input.uniDI.stEbusDI.EL1889_01.DI1 <-> Channel 1/Input
//     ModbusTask Inputs/GVL_Input.uniDI.stEbusDI.EL1889_01.DI10 <-> Channel 10/Input
//     ModbusTask Inputs/GVL_Input.uniDI.stEbusDI.EL1889_01.DI11 <-> Channel 11/Input
//     ModbusTask Inputs/GVL_Input.uniDI.stEbusDI.EL1889_01.DI12 <-> Channel 12/Input
//     ModbusTask Inputs/GVL_Input.uniDI.stEbusDI.EL1889_01.DI13 <-> Channel 13/Input
//     ModbusTask Inputs/GVL_Input.uniDI.stEbusDI.EL1889_01.DI14 <-> Channel 14/Input
//     ModbusTask Inputs/GVL_Input.uniDI.stEbusDI.EL1889_01.DI15 <-> Channel 15/Input
//     ModbusTask Inputs/GVL_Input.uniDI.stEbusDI.EL1889_01.DI16 <-> Channel 16/Input
//     ModbusTask Inputs/GVL_Input.uniDI.stEbusDI.EL1889_01.DI2 <-> Channel 2/Input
//     ModbusTask Inputs/GVL_Input.uniDI.stEbusDI.EL1889_01.DI3 <-> Channel 3/Input
//     ModbusTask Inputs/GVL_Input.uniDI.stEbusDI.EL1889_01.DI4 <-> Channel 4/Input
//     ModbusTask Inputs/GVL_Input.uniDI.stEbusDI.EL1889_01.DI5 <-> Channel 5/Input
//     ModbusTask Inputs/GVL_Input.uniDI.stEbusDI.EL1889_01.DI6 <-> Channel 6/Input
//     ModbusTask Inputs/GVL_Input.uniDI.stEbusDI.EL1889_01.DI7 <-> Channel 7/Input
//     ModbusTask Inputs/GVL_Input.uniDI.stEbusDI.EL1889_01.DI8 <-> Channel 8/Input
//     ModbusTask Inputs/GVL_Input.uniDI.stEbusDI.EL1889_01.DI9 <-> Channel 9/Input
//   DAS_CoreSys/DAS_CoreSys Instance <-> Device 1 (EtherCAT) Storage/Term 1 (EK1200)/Term 7 (EL1889)_02(X7)
//     ModbusTask Inputs/GVL_Input.uniDI.stEbusDI.EL1889_02.DI1 <-> Channel 1/Input
//     ModbusTask Inputs/GVL_Input.uniDI.stEbusDI.EL1889_02.DI10 <-> Channel 10/Input
//     ModbusTask Inputs/GVL_Input.uniDI.stEbusDI.EL1889_02.DI11 <-> Channel 11/Input
//     ModbusTask Inputs/GVL_Input.uniDI.stEbusDI.EL1889_02.DI12 <-> Channel 12/Input
//     ModbusTask Inputs/GVL_Input.uniDI.stEbusDI.EL1889_02.DI13 <-> Channel 13/Input
//     ModbusTask Inputs/GVL_Input.uniDI.stEbusDI.EL1889_02.DI14 <-> Channel 14/Input
//     ModbusTask Inputs/GVL_Input.uniDI.stEbusDI.EL1889_02.DI15 <-> Channel 15/Input
//     ModbusTask Inputs/GVL_Input.uniDI.stEbusDI.EL1889_02.DI16 <-> Channel 16/Input
//     ModbusTask Inputs/GVL_Input.uniDI.stEbusDI.EL1889_02.DI2 <-> Channel 2/Input
//     ModbusTask Inputs/GVL_Input.uniDI.stEbusDI.EL1889_02.DI3 <-> Channel 3/Input
//     ModbusTask Inputs/GVL_Input.uniDI.stEbusDI.EL1889_02.DI4 <-> Channel 4/Input
//     ModbusTask Inputs/GVL_Input.uniDI.stEbusDI.EL1889_02.DI5 <-> Channel 5/Input
//     ModbusTask Inputs/GVL_Input.uniDI.stEbusDI.EL1889_02.DI6 <-> Channel 6/Input
//     ModbusTask Inputs/GVL_Input.uniDI.stEbusDI.EL1889_02.DI7 <-> Channel 7/Input
//     ModbusTask Inputs/GVL_Input.uniDI.stEbusDI.EL1889_02.DI8 <-> Channel 8/Input
//     ModbusTask Inputs/GVL_Input.uniDI.stEbusDI.EL1889_02.DI9 <-> Channel 9/Input
//   DAS_CoreSys/DAS_CoreSys Instance <-> Device 1 (EtherCAT) Storage/Term 1 (EK1200)/Term 8 (EL1889)_03(X9)
//     ModbusTask Inputs/GVL_Input.uniDI.stEbusDI.EL1889_03.DI1 <-> Channel 1/Input
//     ModbusTask Inputs/GVL_Input.uniDI.stEbusDI.EL1889_03.DI10 <-> Channel 10/Input
//     ModbusTask Inputs/GVL_Input.uniDI.stEbusDI.EL1889_03.DI11 <-> Channel 11/Input
//     ModbusTask Inputs/GVL_Input.uniDI.stEbusDI.EL1889_03.DI12 <-> Channel 12/Input
//     ModbusTask Inputs/GVL_Input.uniDI.stEbusDI.EL1889_03.DI13 <-> Channel 13/Input
//     ModbusTask Inputs/GVL_Input.uniDI.stEbusDI.EL1889_03.DI14 <-> Channel 14/Input
//     ModbusTask Inputs/GVL_Input.uniDI.stEbusDI.EL1889_03.DI15 <-> Channel 15/Input
//     ModbusTask Inputs/GVL_Input.uniDI.stEbusDI.EL1889_03.DI16 <-> Channel 16/Input
//     ModbusTask Inputs/GVL_Input.uniDI.stEbusDI.EL1889_03.DI2 <-> Channel 2/Input
//     ModbusTask Inputs/GVL_Input.uniDI.stEbusDI.EL1889_03.DI3 <-> Channel 3/Input
//     ModbusTask Inputs/GVL_Input.uniDI.stEbusDI.EL1889_03.DI4 <-> Channel 4/Input
//     ModbusTask Inputs/GVL_Input.uniDI.stEbusDI.EL1889_03.DI5 <-> Channel 5/Input
//     ModbusTask Inputs/GVL_Input.uniDI.stEbusDI.EL1889_03.DI6 <-> Channel 6/Input
//     ModbusTask Inputs/GVL_Input.uniDI.stEbusDI.EL1889_03.DI7 <-> Channel 7/Input
//     ModbusTask Inputs/GVL_Input.uniDI.stEbusDI.EL1889_03.DI8 <-> Channel 8/Input
//     ModbusTask Inputs/GVL_Input.uniDI.stEbusDI.EL1889_03.DI9 <-> Channel 9/Input
//   DAS_CoreSys/DAS_CoreSys Instance <-> Device 1 (EtherCAT) Storage/Term 1 (EK1200)/Term 9 (EL1889)_04(X10)
//     ModbusTask Inputs/GVL_Input.uniDI.stEbusDI.EL1889_04.DI1 <-> Channel 1/Input
//     ModbusTask Inputs/GVL_Input.uniDI.stEbusDI.EL1889_04.DI10 <-> Channel 10/Input
//     ModbusTask Inputs/GVL_Input.uniDI.stEbusDI.EL1889_04.DI11 <-> Channel 11/Input
//     ModbusTask Inputs/GVL_Input.uniDI.stEbusDI.EL1889_04.DI12 <-> Channel 12/Input
//     ModbusTask Inputs/GVL_Input.uniDI.stEbusDI.EL1889_04.DI13 <-> Channel 13/Input
//     ModbusTask Inputs/GVL_Input.uniDI.stEbusDI.EL1889_04.DI14 <-> Channel 14/Input
//     ModbusTask Inputs/GVL_Input.uniDI.stEbusDI.EL1889_04.DI15 <-> Channel 15/Input
//     ModbusTask Inputs/GVL_Input.uniDI.stEbusDI.EL1889_04.DI16 <-> Channel 16/Input
//     ModbusTask Inputs/GVL_Input.uniDI.stEbusDI.EL1889_04.DI2 <-> Channel 2/Input
//     ModbusTask Inputs/GVL_Input.uniDI.stEbusDI.EL1889_04.DI3 <-> Channel 3/Input
//     ModbusTask Inputs/GVL_Input.uniDI.stEbusDI.EL1889_04.DI4 <-> Channel 4/Input
//     ModbusTask Inputs/GVL_Input.uniDI.stEbusDI.EL1889_04.DI5 <-> Channel 5/Input
//     ModbusTask Inputs/GVL_Input.uniDI.stEbusDI.EL1889_04.DI6 <-> Channel 6/Input
//     ModbusTask Inputs/GVL_Input.uniDI.stEbusDI.EL1889_04.DI7 <-> Channel 7/Input
//     ModbusTask Inputs/GVL_Input.uniDI.stEbusDI.EL1889_04.DI8 <-> Channel 8/Input
//     ModbusTask Inputs/GVL_Input.uniDI.stEbusDI.EL1889_04.DI9 <-> Channel 9/Input
//   DAS_CoreSys/DAS_CoreSys Instance <-> Device 4 (EtherCAT) Allocate/Term 22 (EK1100)/Term 23 (EL1889)_05(X0)
//     ModbusTask Inputs/GVL_Input.uniDI.stEbusDI.EL1889_05.DI1 <-> Channel 1/Input
//     ModbusTask Inputs/GVL_Input.uniDI.stEbusDI.EL1889_05.DI10 <-> Channel 10/Input
//     ModbusTask Inputs/GVL_Input.uniDI.stEbusDI.EL1889_05.DI11 <-> Channel 11/Input
//     ModbusTask Inputs/GVL_Input.uniDI.stEbusDI.EL1889_05.DI12 <-> Channel 12/Input
//     ModbusTask Inputs/GVL_Input.uniDI.stEbusDI.EL1889_05.DI13 <-> Channel 13/Input
//     ModbusTask Inputs/GVL_Input.uniDI.stEbusDI.EL1889_05.DI14 <-> Channel 14/Input
//     ModbusTask Inputs/GVL_Input.uniDI.stEbusDI.EL1889_05.DI15 <-> Channel 15/Input
//     ModbusTask Inputs/GVL_Input.uniDI.stEbusDI.EL1889_05.DI16 <-> Channel 16/Input
//     ModbusTask Inputs/GVL_Input.uniDI.stEbusDI.EL1889_05.DI2 <-> Channel 2/Input
//     ModbusTask Inputs/GVL_Input.uniDI.stEbusDI.EL1889_05.DI3 <-> Channel 3/Input
//     ModbusTask Inputs/GVL_Input.uniDI.stEbusDI.EL1889_05.DI4 <-> Channel 4/Input
//     ModbusTask Inputs/GVL_Input.uniDI.stEbusDI.EL1889_05.DI5 <-> Channel 5/Input
//     ModbusTask Inputs/GVL_Input.uniDI.stEbusDI.EL1889_05.DI6 <-> Channel 6/Input
//     ModbusTask Inputs/GVL_Input.uniDI.stEbusDI.EL1889_05.DI7 <-> Channel 7/Input
//     ModbusTask Inputs/GVL_Input.uniDI.stEbusDI.EL1889_05.DI8 <-> Channel 8/Input
//     ModbusTask Inputs/GVL_Input.uniDI.stEbusDI.EL1889_05.DI9 <-> Channel 9/Input
//   DAS_CoreSys/DAS_CoreSys Instance <-> Device 4 (EtherCAT) Allocate/Term 22 (EK1100)/Term 24 (EL1889)_06(X1)
//     ModbusTask Inputs/GVL_Input.uniDI.stEbusDI.EL1889_06.DI1 <-> Channel 1/Input
//     ModbusTask Inputs/GVL_Input.uniDI.stEbusDI.EL1889_06.DI10 <-> Channel 10/Input
//     ModbusTask Inputs/GVL_Input.uniDI.stEbusDI.EL1889_06.DI11 <-> Channel 11/Input
//     ModbusTask Inputs/GVL_Input.uniDI.stEbusDI.EL1889_06.DI12 <-> Channel 12/Input
//     ModbusTask Inputs/GVL_Input.uniDI.stEbusDI.EL1889_06.DI13 <-> Channel 13/Input
//     ModbusTask Inputs/GVL_Input.uniDI.stEbusDI.EL1889_06.DI14 <-> Channel 14/Input
//     ModbusTask Inputs/GVL_Input.uniDI.stEbusDI.EL1889_06.DI15 <-> Channel 15/Input
//     ModbusTask Inputs/GVL_Input.uniDI.stEbusDI.EL1889_06.DI16 <-> Channel 16/Input
//     ModbusTask Inputs/GVL_Input.uniDI.stEbusDI.EL1889_06.DI2 <-> Channel 2/Input
//     ModbusTask Inputs/GVL_Input.uniDI.stEbusDI.EL1889_06.DI3 <-> Channel 3/Input
//     ModbusTask Inputs/GVL_Input.uniDI.stEbusDI.EL1889_06.DI4 <-> Channel 4/Input
//     ModbusTask Inputs/GVL_Input.uniDI.stEbusDI.EL1889_06.DI5 <-> Channel 5/Input
//     ModbusTask Inputs/GVL_Input.uniDI.stEbusDI.EL1889_06.DI6 <-> Channel 6/Input
//     ModbusTask Inputs/GVL_Input.uniDI.stEbusDI.EL1889_06.DI7 <-> Channel 7/Input
//     ModbusTask Inputs/GVL_Input.uniDI.stEbusDI.EL1889_06.DI8 <-> Channel 8/Input
//     ModbusTask Inputs/GVL_Input.uniDI.stEbusDI.EL1889_06.DI9 <-> Channel 9/Input
//   DAS_CoreSys/DAS_CoreSys Instance <-> Device 4 (EtherCAT) Allocate/Term 22 (EK1100)/Term 25 (EL1889)_07(X2)
//     ModbusTask Inputs/GVL_Input.uniDI.stEbusDI.EL1889_07.DI1 <-> Channel 1/Input
//     ModbusTask Inputs/GVL_Input.uniDI.stEbusDI.EL1889_07.DI10 <-> Channel 10/Input
//     ModbusTask Inputs/GVL_Input.uniDI.stEbusDI.EL1889_07.DI11 <-> Channel 11/Input
//     ModbusTask Inputs/GVL_Input.uniDI.stEbusDI.EL1889_07.DI12 <-> Channel 12/Input
//     ModbusTask Inputs/GVL_Input.uniDI.stEbusDI.EL1889_07.DI13 <-> Channel 13/Input
//     ModbusTask Inputs/GVL_Input.uniDI.stEbusDI.EL1889_07.DI14 <-> Channel 14/Input
//     ModbusTask Inputs/GVL_Input.uniDI.stEbusDI.EL1889_07.DI15 <-> Channel 15/Input
//     ModbusTask Inputs/GVL_Input.uniDI.stEbusDI.EL1889_07.DI16 <-> Channel 16/Input
//     ModbusTask Inputs/GVL_Input.uniDI.stEbusDI.EL1889_07.DI2 <-> Channel 2/Input
//     ModbusTask Inputs/GVL_Input.uniDI.stEbusDI.EL1889_07.DI3 <-> Channel 3/Input
//     ModbusTask Inputs/GVL_Input.uniDI.stEbusDI.EL1889_07.DI4 <-> Channel 4/Input
//     ModbusTask Inputs/GVL_Input.uniDI.stEbusDI.EL1889_07.DI5 <-> Channel 5/Input
//     ModbusTask Inputs/GVL_Input.uniDI.stEbusDI.EL1889_07.DI6 <-> Channel 6/Input
//     ModbusTask Inputs/GVL_Input.uniDI.stEbusDI.EL1889_07.DI7 <-> Channel 7/Input
//     ModbusTask Inputs/GVL_Input.uniDI.stEbusDI.EL1889_07.DI8 <-> Channel 8/Input
//     ModbusTask Inputs/GVL_Input.uniDI.stEbusDI.EL1889_07.DI9 <-> Channel 9/Input
//   DAS_CoreSys/DAS_CoreSys Instance <-> Device 4 (EtherCAT) Allocate/Term 22 (EK1100)/Term 26 (EL1889)_08(X3)
//     ModbusTask Inputs/GVL_Input.uniDI.stEbusDI.EL1889_08.DI1 <-> Channel 1/Input
//     ModbusTask Inputs/GVL_Input.uniDI.stEbusDI.EL1889_08.DI10 <-> Channel 10/Input
//     ModbusTask Inputs/GVL_Input.uniDI.stEbusDI.EL1889_08.DI11 <-> Channel 11/Input
//     ModbusTask Inputs/GVL_Input.uniDI.stEbusDI.EL1889_08.DI12 <-> Channel 12/Input
//     ModbusTask Inputs/GVL_Input.uniDI.stEbusDI.EL1889_08.DI13 <-> Channel 13/Input
//     ModbusTask Inputs/GVL_Input.uniDI.stEbusDI.EL1889_08.DI14 <-> Channel 14/Input
//     ModbusTask Inputs/GVL_Input.uniDI.stEbusDI.EL1889_08.DI15 <-> Channel 15/Input
//     ModbusTask Inputs/GVL_Input.uniDI.stEbusDI.EL1889_08.DI16 <-> Channel 16/Input
//     ModbusTask Inputs/GVL_Input.uniDI.stEbusDI.EL1889_08.DI2 <-> Channel 2/Input
//     ModbusTask Inputs/GVL_Input.uniDI.stEbusDI.EL1889_08.DI3 <-> Channel 3/Input
//     ModbusTask Inputs/GVL_Input.uniDI.stEbusDI.EL1889_08.DI4 <-> Channel 4/Input
//     ModbusTask Inputs/GVL_Input.uniDI.stEbusDI.EL1889_08.DI5 <-> Channel 5/Input
//     ModbusTask Inputs/GVL_Input.uniDI.stEbusDI.EL1889_08.DI6 <-> Channel 6/Input
//     ModbusTask Inputs/GVL_Input.uniDI.stEbusDI.EL1889_08.DI7 <-> Channel 7/Input
//     ModbusTask Inputs/GVL_Input.uniDI.stEbusDI.EL1889_08.DI8 <-> Channel 8/Input
//     ModbusTask Inputs/GVL_Input.uniDI.stEbusDI.EL1889_08.DI9 <-> Channel 9/Input
//   DAS_CoreSys/DAS_CoreSys Instance <-> Device 4 (EtherCAT) Allocate/Term 22 (EK1100)/Term 27 (EL1889)_09(X8)
//     ModbusTask Inputs/GVL_Input.uniDI.stEbusDI.EL1889_09.DI1 <-> Channel 1/Input
//     ModbusTask Inputs/GVL_Input.uniDI.stEbusDI.EL1889_09.DI10 <-> Channel 10/Input
//     ModbusTask Inputs/GVL_Input.uniDI.stEbusDI.EL1889_09.DI11 <-> Channel 11/Input
//     ModbusTask Inputs/GVL_Input.uniDI.stEbusDI.EL1889_09.DI12 <-> Channel 12/Input
//     ModbusTask Inputs/GVL_Input.uniDI.stEbusDI.EL1889_09.DI13 <-> Channel 13/Input
//     ModbusTask Inputs/GVL_Input.uniDI.stEbusDI.EL1889_09.DI14 <-> Channel 14/Input
//     ModbusTask Inputs/GVL_Input.uniDI.stEbusDI.EL1889_09.DI15 <-> Channel 15/Input
//     ModbusTask Inputs/GVL_Input.uniDI.stEbusDI.EL1889_09.DI16 <-> Channel 16/Input
//     ModbusTask Inputs/GVL_Input.uniDI.stEbusDI.EL1889_09.DI2 <-> Channel 2/Input
//     ModbusTask Inputs/GVL_Input.uniDI.stEbusDI.EL1889_09.DI3 <-> Channel 3/Input
//     ModbusTask Inputs/GVL_Input.uniDI.stEbusDI.EL1889_09.DI4 <-> Channel 4/Input
//     ModbusTask Inputs/GVL_Input.uniDI.stEbusDI.EL1889_09.DI5 <-> Channel 5/Input
//     ModbusTask Inputs/GVL_Input.uniDI.stEbusDI.EL1889_09.DI6 <-> Channel 6/Input
//     ModbusTask Inputs/GVL_Input.uniDI.stEbusDI.EL1889_09.DI7 <-> Channel 7/Input
//     ModbusTask Inputs/GVL_Input.uniDI.stEbusDI.EL1889_09.DI8 <-> Channel 8/Input
//     ModbusTask Inputs/GVL_Input.uniDI.stEbusDI.EL1889_09.DI9 <-> Channel 9/Input
//   DAS_CoreSys/DAS_CoreSys Instance <-> Device 4 (EtherCAT) Allocate/Term 22 (EK1100)/Term 28 (EL1889)_10(X11)
//     ModbusTask Inputs/GVL_Input.uniDI.stEbusDI.EL1889_10.DI{1..16} <-> Channel {1..16}/Input  (16 links)
//   DAS_CoreSys/DAS_CoreSys Instance <-> Device 4 (EtherCAT) Allocate/Term 22 (EK1100)/Term 29 (EL2889)_08(Y0)
//     ModbusTask Outputs/GVL_Output.uniDO.stEbusDO.EL2889_08.DO1 <-> Channel 1/Output
//     ModbusTask Outputs/GVL_Output.uniDO.stEbusDO.EL2889_08.DO10 <-> Channel 10/Output
//     ModbusTask Outputs/GVL_Output.uniDO.stEbusDO.EL2889_08.DO11 <-> Channel 11/Output
//     ModbusTask Outputs/GVL_Output.uniDO.stEbusDO.EL2889_08.DO12 <-> Channel 12/Output
//     ModbusTask Outputs/GVL_Output.uniDO.stEbusDO.EL2889_08.DO13 <-> Channel 13/Output
//     ModbusTask Outputs/GVL_Output.uniDO.stEbusDO.EL2889_08.DO14 <-> Channel 14/Output
//     ModbusTask Outputs/GVL_Output.uniDO.stEbusDO.EL2889_08.DO15 <-> Channel 15/Output
//     ModbusTask Outputs/GVL_Output.uniDO.stEbusDO.EL2889_08.DO16 <-> Channel 16/Output
//     ModbusTask Outputs/GVL_Output.uniDO.stEbusDO.EL2889_08.DO2 <-> Channel 2/Output
//     ModbusTask Outputs/GVL_Output.uniDO.stEbusDO.EL2889_08.DO3 <-> Channel 3/Output
//     ModbusTask Outputs/GVL_Output.uniDO.stEbusDO.EL2889_08.DO4 <-> Channel 4/Output
//     ModbusTask Outputs/GVL_Output.uniDO.stEbusDO.EL2889_08.DO5 <-> Channel 5/Output
//     ModbusTask Outputs/GVL_Output.uniDO.stEbusDO.EL2889_08.DO6 <-> Channel 6/Output
//     ModbusTask Outputs/GVL_Output.uniDO.stEbusDO.EL2889_08.DO7 <-> Channel 7/Output
//     ModbusTask Outputs/GVL_Output.uniDO.stEbusDO.EL2889_08.DO8 <-> Channel 8/Output
//     ModbusTask Outputs/GVL_Output.uniDO.stEbusDO.EL2889_08.DO9 <-> Channel 9/Output
//   DAS_CoreSys/DAS_CoreSys Instance <-> Device 4 (EtherCAT) Allocate/Term 22 (EK1100)/Term 30 (EL2889)_09(Y1)
//     ModbusTask Outputs/GVL_Output.uniDO.stEbusDO.EL2889_09.DO1 <-> Channel 1/Output
//     ModbusTask Outputs/GVL_Output.uniDO.stEbusDO.EL2889_09.DO10 <-> Channel 10/Output
//     ModbusTask Outputs/GVL_Output.uniDO.stEbusDO.EL2889_09.DO11 <-> Channel 11/Output
//     ModbusTask Outputs/GVL_Output.uniDO.stEbusDO.EL2889_09.DO12 <-> Channel 12/Output
//     ModbusTask Outputs/GVL_Output.uniDO.stEbusDO.EL2889_09.DO13 <-> Channel 13/Output
//     ModbusTask Outputs/GVL_Output.uniDO.stEbusDO.EL2889_09.DO14 <-> Channel 14/Output
//     ModbusTask Outputs/GVL_Output.uniDO.stEbusDO.EL2889_09.DO15 <-> Channel 15/Output
//     ModbusTask Outputs/GVL_Output.uniDO.stEbusDO.EL2889_09.DO16 <-> Channel 16/Output
//     ModbusTask Outputs/GVL_Output.uniDO.stEbusDO.EL2889_09.DO2 <-> Channel 2/Output
//     ModbusTask Outputs/GVL_Output.uniDO.stEbusDO.EL2889_09.DO3 <-> Channel 3/Output
//     ModbusTask Outputs/GVL_Output.uniDO.stEbusDO.EL2889_09.DO4 <-> Channel 4/Output
//     ModbusTask Outputs/GVL_Output.uniDO.stEbusDO.EL2889_09.DO5 <-> Channel 5/Output
//     ModbusTask Outputs/GVL_Output.uniDO.stEbusDO.EL2889_09.DO6 <-> Channel 6/Output
//     ModbusTask Outputs/GVL_Output.uniDO.stEbusDO.EL2889_09.DO7 <-> Channel 7/Output
//     ModbusTask Outputs/GVL_Output.uniDO.stEbusDO.EL2889_09.DO8 <-> Channel 8/Output
//     ModbusTask Outputs/GVL_Output.uniDO.stEbusDO.EL2889_09.DO9 <-> Channel 9/Output
//   DAS_CoreSys/DAS_CoreSys Instance <-> Device 4 (EtherCAT) Allocate/Term 22 (EK1100)/Term 31 (EL2889)_10(Y2)
//     ModbusTask Outputs/GVL_Output.uniDO.stEbusDO.EL2889_10.DO{1..16} <-> Channel {1..16}/Output  (16 links)
//   DAS_CoreSys/DAS_CoreSys Instance <-> Device 4 (EtherCAT) Allocate/Term 22 (EK1100)/Term 33 (EL1889)_11(X4)
//     ModbusTask Inputs/GVL_Input.uniDI.stEbusDI.EL1889_11.DI{1..16} <-> Channel {1..16}/Input  (16 links)
//   DAS_CoreSys/DAS_CoreSys Instance <-> Device 6 (ECAT EIP Scanner (EL6652))
//     CoreSys Inputs/DAS_CoreSys.MachineControl.FanucRobot.List.ShippingRobot._FanucEIPState <-> Inputs/ECatState
//   DAS_CoreSys/DAS_CoreSys Instance <-> Device 6 (ECAT EIP Scanner (EL6652))/FANUC Robot R30iB+
//     CoreSys Inputs/DAS_CoreSys.MachineControl.FanucRobot.List.ShippingRobot._EIPConnectionState <-> Inputs/State
//     CoreSys Inputs/DAS_CoreSys.MachineControl.FanucRobot.List.ShippingRobot._rawIn_DI <-> DIO (Input/Output)/Inputs/noname0_arrBYTE
//     CoreSys Inputs/DAS_CoreSys.MachineControl.FanucRobot.List.ShippingRobot._rawIn_UI <-> UIO (Input/Output)/Inputs/noname0_arrBYTE
//     CoreSys Outputs/DAS_CoreSys.MachineControl.FanucRobot.List.ShippingRobot._rawOut_DO <-> DIO (Input/Output)/Outputs/noname0_arrBYTE
//     CoreSys Outputs/DAS_CoreSys.MachineControl.FanucRobot.List.ShippingRobot._rawOut_UO <-> UIO (Input/Output)/Outputs/noname0_arrBYTE
//   DAS_CoreSys/DAS_CoreSys Instance <-> Storage Fanuc Robot (ECAT EIP Scanner (EL6652))
//     CoreSys Inputs/DAS_CoreSys.MachineControl.FanucRobot.List.StorageRobot._FanucEIPState <-> Inputs/ECatState
//   DAS_CoreSys/DAS_CoreSys Instance <-> Storage Fanuc Robot (ECAT EIP Scanner (EL6652))/FANUC Robot R30iB+
//     CoreSys Inputs/DAS_CoreSys.MachineControl.FanucRobot.List.StorageRobot._EIPConnectionState <-> Inputs/State
//     CoreSys Inputs/DAS_CoreSys.MachineControl.FanucRobot.List.StorageRobot._rawIn_DI <-> DIO (Input/Output)/Inputs/noname0_arrBYTE
//     CoreSys Inputs/DAS_CoreSys.MachineControl.FanucRobot.List.StorageRobot._rawIn_UI <-> UIO (Input/Output)/Inputs/noname0_arrBYTE
//     CoreSys Outputs/DAS_CoreSys.MachineControl.FanucRobot.List.StorageRobot._rawOut_DO <-> DIO (Input/Output)/Outputs/noname0_arrBYTE
//     CoreSys Outputs/DAS_CoreSys.MachineControl.FanucRobot.List.StorageRobot._rawOut_UO <-> UIO (Input/Output)/Outputs/noname0_arrBYTE
//   DAS_CoreSys/DAS_CoreSys Instance <-> NC-Task 1 SAF/Axes/Axis 1|TurnTable
//     MotionSync Inputs/BATW.GVL_Motion.arAxisCtrl_gb[1].Admin.Axis.NcToPlc <-> Outputs/ToPlc
//     MotionSync Outputs/BATW.GVL_Motion.arAxisCtrl_gb[1].Admin.Axis.PlcToNc <-> Inputs/FromPlc
//   DAS_CoreSys/DAS_CoreSys Instance <-> NC-Task 1 SAF/Axes/Axis 2|RoundBelt
//     MotionSync Inputs/BATW.GVL_Motion.arAxisCtrl_gb[2].Admin.Axis.NcToPlc <-> Outputs/ToPlc
//     MotionSync Outputs/BATW.GVL_Motion.arAxisCtrl_gb[2].Admin.Axis.PlcToNc <-> Inputs/FromPlc
//   DAS_CoreSys/DAS_CoreSys Instance <-> NC-Task 1 SAF/Axes/Axis 3|AllocateRobot_X
//     MotionSync Inputs/BATW.GVL_Motion.arAxisCtrl_gb[3].Admin.Axis.NcToPlc <-> Outputs/ToPlc
//     MotionSync Outputs/BATW.GVL_Motion.arAxisCtrl_gb[3].Admin.Axis.PlcToNc <-> Inputs/FromPlc
//   DAS_CoreSys/DAS_CoreSys Instance <-> NC-Task 1 SAF/Axes/Axis 4|AllocateRobot_Y
//     MotionSync Inputs/BATW.GVL_Motion.arAxisCtrl_gb[4].Admin.Axis.NcToPlc <-> Outputs/ToPlc
//     MotionSync Outputs/BATW.GVL_Motion.arAxisCtrl_gb[4].Admin.Axis.PlcToNc <-> Inputs/FromPlc
//   DAS_CoreSys/DAS_CoreSys Instance <-> NC-Task 1 SAF/Axes/Axis 5|OutRobot_X
//     MotionSync Inputs/BATW.GVL_Motion.arAxisCtrl_gb[5].Admin.Axis.NcToPlc <-> Outputs/ToPlc
//     MotionSync Outputs/BATW.GVL_Motion.arAxisCtrl_gb[5].Admin.Axis.PlcToNc <-> Inputs/FromPlc
//   DAS_CoreSys/DAS_CoreSys Instance <-> NC-Task 1 SAF/Axes/Axis 6|OutRobot_Y
//     MotionSync Inputs/BATW.GVL_Motion.arAxisCtrl_gb[6].Admin.Axis.NcToPlc <-> Outputs/ToPlc
//     MotionSync Outputs/BATW.GVL_Motion.arAxisCtrl_gb[6].Admin.Axis.PlcToNc <-> Inputs/FromPlc
//   DAS_CoreSys/DAS_CoreSys Instance <-> NC-Task 1 SAF/Axes/Axis 7|RackMotor
//     MotionSync Inputs/BATW.GVL_Motion.arAxisCtrl_gb[7].Admin.Axis.NcToPlc <-> Outputs/ToPlc
//     MotionSync Outputs/BATW.GVL_Motion.arAxisCtrl_gb[7].Admin.Axis.PlcToNc <-> Inputs/FromPlc

CONFIGURATION DAS_CoreSys
    RESOURCE PLC ON TwinCAT3
        TASK CoreSys(INTERVAL := T#10ms, PRIORITY := 20);
        TASK ModbusTask(INTERVAL := T#5ms, PRIORITY := 21);
        TASK MotionSync(INTERVAL := T#2ms, PRIORITY := 1);
        PROGRAM ComModbusRTU WITH CoreSys : ComModbusRTU;
        PROGRAM DAS_CoreSys WITH CoreSys : DAS_CoreSys;
        PROGRAM ComModbusRTU WITH ModbusTask : ComModbusRTU;
        PROGRAM DAS_MotionSync WITH MotionSync : DAS_MotionSync;
    END_RESOURCE
END_CONFIGURATION

// ---- Library/00_PackML/01_ObjectBase/eModeChangeState.TcDUT
{attribute 'qualified_only'}
{attribute 'strict'}
TYPE eModeChangeState :
(
	WaitingRequest := 0, // Waiting for user request
	StartingUnitModeManager := 1, // Execute unit manager
	ErrorHandling :=2 // After execute, check unit manager status
);
END_TYPE

// ---- Library/00_PackML/02_Mode/E_Severity.TcDUT
{attribute 'qualified_only'}
TYPE E_Severity :
(
	// No define or form subsys issue
	Disregard := 0,
	// Level1 Subsys Error or normal alarm
	Level1,
	// Level2 Set Held -> normal error
	Level2,
	Level3,
	Level4,
	Level5,
	// Level6 Set Held -> XTS
	Level6, 
	// Level7 Set Aobrt
	Level7 := 7
)DINT;
END_TYPE

// ---- Library/00_PackML/02_Mode/E_UnitMode.TcDUT
{attribute 'qualified_only'}
TYPE E_UnitMode :
(
        Undefined   := 0, // Mode not defined.
        Auto        := 1, // Mode Auto, production...
        Manual      := 3, // Mode Manual, user manual control
        Homing      := 4 // Mode Homing, unit's home
)DINT;
END_TYPE

// ---- Library/10_Machine/12_MachineControl/DUTs/AxisNo.TcDUT
{attribute 'qualified_only'}
{attribute 'strict'}
TYPE
    AxisNo :
    (
        TurnTable := 1,
        RoundBelt := 2,
        Allocate_X := 3,
        Allocate_Y := 4,
        OutRobot_X := 5,
        OutRobot_Y := 6,
        RackMotor := 7
    ) UDINT;
END_TYPE

// ---- Library/10_Machine/12_MachineControl/DUTs/Cylinders/ST_CylinderList.TcDUT
TYPE
    ST_CylinderList :
    STRUCT
        fbUpCV_FeedInPress1             : FB_Cylinder;
        fbUpCV_FeedInPress2             : FB_Cylinder;
        fbUpCV_DiameterPress            : FB_Cylinder;
        fbUpCV_CamaraPress1             : FB_Cylinder;
        fbUpCV_CamaraPress2             : FB_Cylinder;
        fbUpCV_CamaraPress3             : FB_Cylinder;
        fbUpCV_CamaraPress4             : FB_Cylinder;
        fbUpCV_Block1                   : FB_Cylinder;
        fbUpCV_Block2                   : FB_Cylinder;
        fbUpCV_Block3                   : FB_Cylinder;
        fbUpCV_DiameterHoriz            : FB_Cylinder;
        fbUpCV_DiameterVert             : FB_Cylinder;
        fbUpCV_DiameterClamp            : FB_Cylinder;
        fbStackPush                     : FB_Cylinder;
        fbPullOutCV_AsidePress1         : FB_Cylinder;
        fbPullOutCV_AsidePress2         : FB_Cylinder;
        fbPullOutCV_AsideBlock          : FB_Cylinder;
        fbPullOutCV_BsidePress1         : FB_Cylinder;
        fbPullOutCV_BsidePress2         : FB_Cylinder;
        fbPullOutCV_BsideBlock          : FB_Cylinder;
        fbLowCV_Press1                  : FB_Cylinder;
        fbLowCV_Press2                  : FB_Cylinder;
        fbLowCV_Press3                  : FB_Cylinder;
        fbLowCV_Press4                  : FB_Cylinder;
        fbLowCV_Block1                  : FB_Cylinder;
        fbLowCV_Block2                  : FB_Cylinder;
        fbAllocateRobot_LeftVert1       : FB_Cylinder;
        fbAllocateRobot_LeftVert2       : FB_Cylinder;
        fbAllocateRobot_RightVert1      : FB_Cylinder;
        fbAllocateRobot_RightVert2      : FB_Cylinder;
        fbAllocateRobot_LeftClamp1      : FB_Cylinder;
        fbAllocateRobot_LeftClamp2      : FB_Cylinder;
        fbAllocateRobot_RightClamp1     : FB_Cylinder;
        fbAllocateRobot_RightClamp2     : FB_Cylinder;
        fbRoundBelt_WorkZone_Press      : FB_Cylinder;
        fbRoundBelt_WorkZone_Plug       : FB_Cylinder;
        fbRoundBelt_ChargeZone_Plug     : FB_Cylinder;
        fbRoundBelt_TransmitCVZone_Plug : FB_Cylinder;
        fbOutRobot_AsideVert            : FB_Cylinder;
        fbOutRobot_BsideVert            : FB_Cylinder;
        fbOutRobot_AsideClamp           : FB_Cylinder;
        fbOutRobot_BsideClamp           : FB_Cylinder;
        fbTransmitCV_CamaraHoriz        : FB_Cylinder;
        fbDifferentSizeCV_Press2        : FB_Cylinder;
        fbDifferentSizeCV_Press1        : FB_Cylinder;
        fbDifferentSizeCV_Block1        : FB_Cylinder;
        fbSameSizeCV_Press4             : FB_Cylinder;
        fbSameSizeCV_Press3             : FB_Cylinder;
        fbSameSizeCV_Press2             : FB_Cylinder;
        fbSameSizeCV_Press1             : FB_Cylinder;
        fbSameSizeCV_Block2             : FB_Cylinder;
        fbSameSizeCV_Block1             : FB_Cylinder;
        fbTurntable_Press               : FB_Cylinder;
    END_STRUCT
END_TYPE

// ---- Library/10_Machine/12_MachineControl/DUTs/Cylinders/UNI_CylinderList.TcDUT
TYPE
    UNI_CylinderList :
    UNION
        arCylinder : ARRAY[1..udiMax_CylinderNum] OF FB_Cylinder;
        List       : ST_CylinderList;
    END_UNION
END_TYPE

// ---- Library/10_Machine/12_MachineControl/DUTs/E_DataFrom.TcDUT
{attribute 'qualified_only'}
{attribute 'strict'}
TYPE
    E_DataFrom :
    (
        Local := 0,
        Remote := 1
    );
END_TYPE

// ---- Library/10_Machine/12_MachineControl/DUTs/FanucRobot/ST_FanucRobotList.TcDUT
TYPE
    ST_FanucRobotList :
    STRUCT
        StorageRobot  : FB_FanucRobot_Basic;
        ShippingRobot : FB_FanucRobot_Basic;
    END_STRUCT
END_TYPE

// ---- Library/10_Machine/12_MachineControl/DUTs/FanucRobot/UNI_FanucRobotList.TcDUT
TYPE
    UNI_FanucRobotList :
    UNION
        arFanucRobot : ARRAY[1..2] OF FB_FanucRobot_Basic;
        List         : ST_FanucRobotList;
    END_UNION
END_TYPE

// ---- Library/10_Machine/12_MachineControl/DUTs/Motor/ST_MotorList.TcDUT
TYPE
    ST_MotorList :
    STRUCT
        WareHouseCV_01          : FB_Motor;
        WareHouseCV_02          : FB_Motor;
        WareHouseCV_03          : FB_Motor;
        WareHouseCV_04          : FB_Motor;
        WareHouseCV_05          : FB_Motor;
        WareHouseCV_06          : FB_Motor;
        WareHouseCV_07          : FB_Motor;
        WareHouseCV_08          : FB_Motor;
        WareHouseCV_09          : FB_Motor;
        WareHouseCV_10          : FB_Motor;
        WareHouseCV_11          : FB_Motor;
        WareHouseCV_12          : FB_Motor;
        WareHouseCV_13          : FB_Motor;
        WareHouseCV_14          : FB_Motor;
        WareHouseCV_15          : FB_Motor;
        WareHouseCV_16          : FB_Motor;
        WareHouseCV_17          : FB_Motor;
        WareHouseCV_18          : FB_Motor;
        WareHouseCV_19          : FB_Motor;
        WareHouseCV_20          : FB_Motor;
        UpCV                    : FB_Motor;
        LowCV                   : FB_Motor;
        PullOutCV_A             : FB_Motor;
        PullOutCV_B             : FB_Motor;
        TransmitSameSideCV      : FB_Motor;
        TransmitDifferentSideCV : FB_Motor;
    END_STRUCT
END_TYPE

// ---- Library/10_Machine/12_MachineControl/DUTs/Motor/UNI_MotorList.TcDUT
TYPE
    UNI_MotorList :
    UNION
        arMotor : ARRAY[1..26] OF FB_Motor;
        List    : ST_MotorList;
    END_UNION
END_TYPE

// ---- Library/10_Machine/12_MachineControl/DUTs/Service/ST_ServiceCtrl_Base.TcDUT
TYPE
    ST_ServiceCtrl_Base :
    STRUCT
        Execute : BOOL; // Service Execute
        Abort   : BOOL; // Service Abort
        Reset   : BOOL; // Service Reset
    END_STRUCT
END_TYPE

// ---- Library/10_Machine/12_MachineControl/DUTs/Service/ST_ServiceStatus_Base.TcDUT
TYPE
    ST_ServiceStatus_Base :
    STRUCT
        Busy    : BOOL; // Service is running
        Done    : BOOL; // Service process complete
        Error   : BOOL; // Service Error
        Aborted : BOOL; // Service Aborted
    END_STRUCT
END_TYPE

// ---- Library/10_Machine/12_MachineControl/DUTs/Setup/E_ClipNo.TcDUT
{attribute 'qualified_only'}
{attribute 'strict'}
TYPE
    E_ClipNo :
    (
        A := 0,
        B := 1,
        C := 2,
        D := 3
    );
END_TYPE

// ---- Library/10_Machine/12_MachineControl/DUTs/Setup/ST_AllocateRobotCoordinate.TcDUT
TYPE
    ST_AllocateRobotCoordinate :
    STRUCT
        fname          : STRING;
        index          : LREAL;
        TargetDistance : LREAL;
        Execute        : BOOL; // 沒作用是否刪除?
        Done           : BOOL; // 沒作用是否刪除?
    END_STRUCT
END_TYPE

// ---- Library/10_Machine/12_MachineControl/DUTs/Setup/ST_AllocateRobotPositionTable.TcDUT
TYPE
    ST_AllocateRobotPositionTable :
    STRUCT
    END_STRUCT
END_TYPE

// ---- Library/10_Machine/12_MachineControl/DUTs/Setup/ST_AxisPara.TcDUT
TYPE
    ST_AxisPara :
    STRUCT
        Manual   : ST_AxisPara_Manual; 	// 手動控制參數
        Auto     : ST_AxisPara_Auto; 	// 自動控制參數
        Homing   : ST_AxisPara_Homing; 	// 回HOME參數
    END_STRUCT
END_TYPE

// ---- Library/10_Machine/12_MachineControl/DUTs/Setup/ST_AxisPara_Auto.TcDUT
TYPE
    ST_AxisPara_Auto :
    STRUCT
        Velocity     : LREAL := 10; // The velocity command used during AxisMove in AutoMode within DAS_CoreSys.
        Acceleration : LREAL := 100; // The Acceleration command used during AxisMove in AutoMode within DAS_CoreSys.
        Deceleration : LREAL := 100; // The Deceleration command used during AxisMove in AutoMode within DAS_CoreSys.
        Jerk         : LREAL := 1000; // The Jerk command used during AxisMove in AutoMode within DAS_CoreSys.
    END_STRUCT
END_TYPE

// ---- Library/10_Machine/12_MachineControl/DUTs/Setup/ST_AxisPara_HalfAuto.TcDUT
TYPE
    ST_AxisPara_HalfAuto :
    STRUCT
        Velocity     : LREAL := 10; // The velocity command used during AxisMove in HalfAuto within DAS_CoreSys.
        Acceleration : LREAL := 100; // The Acceleration command used during AxisMove in HalfAuto within DAS_CoreSys.
        Deceleration : LREAL := 100; // The Deceleration command used during AxisMove in HalfAuto within DAS_CoreSys.
        Jerk         : LREAL := 1000; // The Jerk command used during AxisMove in HalfAuto within DAS_CoreSys.
    END_STRUCT
END_TYPE

// ---- Library/10_Machine/12_MachineControl/DUTs/Setup/ST_AxisPara_Homing.TcDUT
TYPE
    ST_AxisPara_Homing :
    STRUCT
        Offset              : LREAL; // after detact home sensor, axis move distance
        SetAbsolutePosition : LREAL; // When homing process completed, set current position according this value.
        FastVelo            : ST_VelocityParameter;
        SlowVelo            : ST_VelocityParameter;

    END_STRUCT
END_TYPE

// ---- Library/10_Machine/12_MachineControl/DUTs/Setup/ST_AxisPara_Manual.TcDUT
TYPE
    ST_AxisPara_Manual :
    STRUCT
        JogVelocity     : LREAL := 10; // According to the unit defined in NC_Parameter, typically mm/s or deg/s.
        JogAcceleration : LREAL := 100; // According to the unit defined in NC_Parameter, typically mm/s^2 or deg/s^2.
        JogDeceleration : LREAL := 100; // According to the unit defined in NC_Parameter, typically mm/s^2 or deg/s^2.
        JogJerk         : LREAL := 1000; // According to the unit defined in NC_Parameter, typically mm/s^3 or deg/s^3.
        PtpVelocity     : LREAL := 10;
        PtpAcceleration : LREAL := 100;
        PtpDeceleration : LREAL := 100;
        PtpJerk         : LREAL := 1000;
        PtpPosition     : LREAL := 0;
    END_STRUCT
END_TYPE

// ---- Library/10_Machine/12_MachineControl/DUTs/Setup/ST_CylinderPara.TcDUT
TYPE
    ST_CylinderPara :
    STRUCT
        ExtendTime       : TIME;
        RetractTime      : TIME;
        ExtendDelayTime  : TIME;
        RetractDelayTime : TIME;
        ExtendOverTime   : TIME;
        RetractOverTime  : TIME;
    END_STRUCT
END_TYPE

// ---- Library/10_Machine/12_MachineControl/DUTs/Setup/ST_FanucRobotCCDSetting.TcDUT
TYPE ST_FanucRobotCCDSetting :
STRUCT
	    WareHouseA_ClampA_UseCCD : BOOL;
        WareHouseA_ClampB_UseCCD : BOOL;
        WareHouseB_ClampA_UseCCD : BOOL;
        WareHouseB_ClampB_UseCCD : BOOL;
        Bzone_UseCCD             : BOOL;
        Czone_UseCCD             : BOOL;
        Dzone_UseCCD             : BOOL;
        Ezone_UseCCD             : BOOL;
        Fzone_UseCCD             : BOOL;
        Gzone_UseCCD             : BOOL;
        Hzone_UseCCD             : BOOL;
        Jzone_UseCCD             : BOOL;
        Kzone_UseCCD             : BOOL;
END_STRUCT
END_TYPE

// ---- Library/10_Machine/12_MachineControl/DUTs/Setup/ST_OutRobotCoordinate.TcDUT
////出料區座標結構
TYPE
    ST_OutRobotCoordinate :
    STRUCT
        fName  : STRING;
        index  : LREAL;
        X      : LREAL;
        Y      : LREAL;
        Rotate : LREAL; // 沒作用是否刪除?
        Clip   : LREAL; // 沒作用是否刪除?
        Excute : BOOL; // 沒作用是否刪除?
        Done   : BOOL; // 沒作用是否刪除?
    END_STRUCT
END_TYPE

// ---- Library/10_Machine/12_MachineControl/DUTs/Setup/ST_OutRobotPositionTable.TcDUT
TYPE
    ST_OutRobotPositionTable :
    STRUCT
    END_STRUCT
END_TYPE

// ---- Library/10_Machine/12_MachineControl/DUTs/Setup/ST_PositionTable.TcDUT
TYPE
    ST_PositionTable :
    STRUCT
        Zone  : STRING;   // 區域
        Index : INT; 	  // 順序
        X_Pos : LREAL; 	  // X-Axis target position (Unit: mm)
        Y_Pos : LREAL; 	  // Y-Axis target position (Unit: mm)
        R_Pos : LREAL; 	  // R-Axis target position (Unit: deg)
        Robot : INT; 	  // 呼叫機器人
        Clip  : E_ClipNo; // 夾爪.
    END_STRUCT
END_TYPE

// ---- Library/10_Machine/12_MachineControl/DUTs/Setup/ST_SetupAxis.TcDUT
TYPE
    ST_SetupAxis :
    STRUCT
        TurnTable  		: ST_AxisPara; 				// 圓盤參數
        Allocate   		: ST_AxisPara; 				// 圓帶參數
        OutRobot_X 		: ST_AxisPara;				// 出料手臂X參數
        OutRobot_Y 		: ST_AxisPara; 				// 出料手臂Y參數
        Needle_X 		: ST_AxisPara; 				// 配針 X參數
        Needle_Y 		: ST_AxisPara; 				// 配針 Y參數
		RackMotor  		: ST_AxisPara; 			    //出貨料架參數
		ElvaterAxis		: ST_AxisPara;				//電梯參數
		HookAxis		: ST_AxisPara;				//勾盤參數
		FinishAxis		: ST_AxisPara;				//出料層架參數
    END_STRUCT
END_TYPE

// ---- Library/10_Machine/12_MachineControl/DUTs/Setup/ST_SetupCylinder.TcDUT
TYPE
    ST_SetupCylinder :
    STRUCT
        UpCV_FeedInPress1             : BATW_Base.ST_CylinderPara;
        UpCV_FeedInPress2             : BATW_Base.ST_CylinderPara;
        UpCV_DiameterPress            : BATW_Base.ST_CylinderPara;
        UpCV_CamaraPress1             : BATW_Base.ST_CylinderPara;
        UpCV_CamaraPress2             : BATW_Base.ST_CylinderPara;
        UpCV_CamaraPress3             : BATW_Base.ST_CylinderPara;
        UpCV_CamaraPress4             : BATW_Base.ST_CylinderPara;
        UpCV_Block1                   : BATW_Base.ST_CylinderPara;
        UpCV_Block2                   : BATW_Base.ST_CylinderPara;
        UpCV_Block3                   : BATW_Base.ST_CylinderPara;
        UpCV_DiameterHoriz            : BATW_Base.ST_CylinderPara;
        UpCV_DiameterVert             : BATW_Base.ST_CylinderPara;
        UpCV_DiameterClamp            : BATW_Base.ST_CylinderPara;
        StackPush                     : BATW_Base.ST_CylinderPara;
        PullOutCV_AsidePress1         : BATW_Base.ST_CylinderPara;
        PullOutCV_AsidePress2         : BATW_Base.ST_CylinderPara;
        PullOutCV_AsideBlock          : BATW_Base.ST_CylinderPara;
        PullOutCV_BsidePress1         : BATW_Base.ST_CylinderPara;
        PullOutCV_BsidePress2         : BATW_Base.ST_CylinderPara;
        PullOutCV_BsideBlock          : BATW_Base.ST_CylinderPara;
        LowCV_Press1                  : BATW_Base.ST_CylinderPara;
        LowCV_Press2                  : BATW_Base.ST_CylinderPara;
        LowCV_Press3                  : BATW_Base.ST_CylinderPara;
        LowCV_Press4                  : BATW_Base.ST_CylinderPara;
        LowCV_Block1                  : BATW_Base.ST_CylinderPara;
        LowCV_Block2                  : BATW_Base.ST_CylinderPara;
        AllocateRobot_LeftVert1       : BATW_Base.ST_CylinderPara;
        AllocateRobot_LeftVert2       : BATW_Base.ST_CylinderPara;
        AllocateRobot_RightVert1      : BATW_Base.ST_CylinderPara;
        AllocateRobot_RightVert2      : BATW_Base.ST_CylinderPara;
        AllocateRobot_LeftClamp1      : BATW_Base.ST_CylinderPara;
        AllocateRobot_LeftClamp2      : BATW_Base.ST_CylinderPara;
        AllocateRobot_RightClamp1     : BATW_Base.ST_CylinderPara;
        AllocateRobot_RightClamp2     : BATW_Base.ST_CylinderPara;
        RoundBelt_WorkZone_Press      : BATW_Base.ST_CylinderPara;
        RoundBelt_WorkZone_Plug       : BATW_Base.ST_CylinderPara;
        RoundBelt_ChargeZone_Plug     : BATW_Base.ST_CylinderPara;
        RoundBelt_TransmitCVZone_Plug : BATW_Base.ST_CylinderPara;
        OutRobot_AsideVert            : BATW_Base.ST_CylinderPara;
        OutRobot_BsideVert            : BATW_Base.ST_CylinderPara;
        OutRobot_AsideClamp           : BATW_Base.ST_CylinderPara;
        OutRobot_BsideClamp           : BATW_Base.ST_CylinderPara;
        TransmitCV_CamaraHoriz        : BATW_Base.ST_CylinderPara;
        DifferentSizeCV_Press2        : BATW_Base.ST_CylinderPara;
        DifferentSizeCV_Press1        : BATW_Base.ST_CylinderPara;
        DifferentSizeCV_Block1        : BATW_Base.ST_CylinderPara;
        SameSizeCV_Press4             : BATW_Base.ST_CylinderPara;
        SameSizeCV_Press3             : BATW_Base.ST_CylinderPara;
        SameSizeCV_Press2             : BATW_Base.ST_CylinderPara;
        SameSizeCV_Press1             : BATW_Base.ST_CylinderPara;
        SameSizeCV_Block2             : BATW_Base.ST_CylinderPara;
        SameSizeCV_Block1             : BATW_Base.ST_CylinderPara;
        Turntable_Press               : BATW_Base.ST_CylinderPara;
    END_STRUCT
END_TYPE

// ---- Library/10_Machine/12_MachineControl/DUTs/Setup/ST_SetupFanucRobot.TcDUT
TYPE
    ST_SetupFanucRobot :
    STRUCT
        RobotVelocity : LREAL :=20;//手臂移動速度百分比
		ZoneCCD : ST_FanucRobotCCDSetting;//CCD使用設定
    END_STRUCT
END_TYPE

// ---- Library/10_Machine/12_MachineControl/DUTs/Setup/ST_SetupMotor.TcDUT
TYPE
    ST_SetupMotor :
    STRUCT
		//A倉軌道
        WareHouseCV_10          : ST_MotorPara;
        WareHouseCV_09          : ST_MotorPara;
        WareHouseCV_08          : ST_MotorPara;
        WareHouseCV_07          : ST_MotorPara;
        WareHouseCV_06          : ST_MotorPara;
        WareHouseCV_05          : ST_MotorPara;
        WareHouseCV_04          : ST_MotorPara;
        WareHouseCV_03          : ST_MotorPara;
        WareHouseCV_02          : ST_MotorPara;
        WareHouseCV_01          : ST_MotorPara;
		//B倉軌道
        WareHouseCV_20          : ST_MotorPara;
        WareHouseCV_19          : ST_MotorPara;
        WareHouseCV_18          : ST_MotorPara;
        WareHouseCV_17          : ST_MotorPara;
        WareHouseCV_16          : ST_MotorPara;
        WareHouseCV_15          : ST_MotorPara;
        WareHouseCV_14          : ST_MotorPara;
        WareHouseCV_13          : ST_MotorPara;
        WareHouseCV_12          : ST_MotorPara;
        WareHouseCV_11          : ST_MotorPara;
		
        UpCV                    : ST_MotorPara;//上層軌道
		
        LowCV                   : ST_MotorPara;//下層軌道
		
        PullOutCV_A             : ST_MotorPara;//空盒軌道
		
        PullOutCV_B             : ST_MotorPara;//待拔針軌道 
		
        TransmitSameSideCV      : ST_MotorPara;//同尺寸軌道
		
        TransmitDifferentSideCV : ST_MotorPara; //配針軌道
    END_STRUCT
END_TYPE

// ---- Library/10_Machine/12_MachineControl/DUTs/Setup/ST_SetupPara.TcDUT
TYPE
    ST_SetupPara :
    STRUCT
        Cylinders     : ST_SetupCylinder;					//汽缸參數
        Axes          : ST_SetupAxis;						//軸參數
        Motor         : ST_SetupMotor;						//軌道參數
        PositionTable : ARRAY[1..200] OF ST_PositionTable;  //點位參數
        StorageRobot  : ST_SetupFanucRobot;					//六軸手臂參數
        Mechanical    : ST_Setup_Mechanical;				//機台參數
	//		Light 		  : ST_Setup_Light;換位子
    END_STRUCT
END_TYPE

// ---- Library/10_Machine/12_MachineControl/DUTs/Setup/ST_Setup_Light.TcDUT
TYPE
    ST_Setup_Light :
    STRUCT
        Storage_EleBoxLight_Off : BOOL; // True : Turn off light
        Storage_AreaLight_Off 	: BOOL; // True : Turn off light
        Allocated_AreaLight_Off : BOOL; //True : Turn off light
    END_STRUCT
END_TYPE

// ---- Library/10_Machine/12_MachineControl/DUTs/Setup/ST_Setup_Mechanical.TcDUT
TYPE
    ST_Setup_Mechanical :
    STRUCT
        //配針手臂在圓帶的盒的左右的間距預設是10
        Allocate_box_leftandRight_Distance 	: LREAL:=10;
        //配針手臂在圓帶的盒的上下的間距預設是10
        Allocate_box_UpandDown_Distance 	: LREAL:=10;  
		// RS485 by pass
		stModbusByPass						:st_ModbusSwitchOff;
		//SafetyDoor
		stSafetyByPass						:st_SafetyByPass;
    END_STRUCT
END_TYPE

// ---- Library/10_Machine/12_MachineControl/DUTs/ST_ChangeIntoProduction.TcDUT
//structure for a visu userwindow, to chnage into productionmode
TYPE
    ST_ChangeIntoProduction :
    STRUCT
        bYes      : BOOL;
        bNo       : BOOL;
        bYesReset : BOOL;
    END_STRUCT
END_TYPE

// ---- Library/10_Machine/12_MachineControl/DUTs/ST_CylinderMonitor.TcDUT
TYPE
    ST_CylinderMonitor :
    STRUCT
        InFrontPosition : BOOL;
        InRearPosition  : BOOL;
        Error           : BOOL;
        ErrMsg          : T_MaxString;
    END_STRUCT
END_TYPE

// ---- Library/10_Machine/12_MachineControl/DUTs/ST_MotorMonitor.TcDUT
TYPE
    ST_MotorMonitor :
    STRUCT
        InForward  : BOOL;
        InBackward : BOOL;
        InStopped  : BOOL;
        Error      : BOOL;
        ErrMsg     : T_MaxString;
    END_STRUCT
END_TYPE

// ---- Library/10_Machine/12_MachineControl/DUTs/ST_TableMoveCtrl.TcDUT
TYPE
    ST_TableMoveCtrl EXTENDS ST_ServiceCtrl_Base :
    STRUCT
        Index : INT; // PositionTable array index
    END_STRUCT
END_TYPE

// ---- Library/10_Machine/12_MachineControl/DUTs/ST_TableMoveService.TcDUT
TYPE
    ST_TableMoveService :
    STRUCT
        Ctrl   : ST_TableMoveCtrl;
        Status : ST_TableMoveStatus;
    END_STRUCT
END_TYPE

// ---- Library/10_Machine/12_MachineControl/DUTs/ST_TableMoveStatus.TcDUT
TYPE
    ST_TableMoveStatus EXTENDS ST_ServiceStatus_Base :
    STRUCT
    END_STRUCT
END_TYPE

// ---- Library/10_Machine/12_MachineControl/DUTs/UnitNo.TcDUT
{attribute 'qualified_only'}
{attribute 'strict'}
TYPE
    UnitNo :
    (
        Machine := 0,
        Storage := 1,
        Allocate := 2,
        Shipping := 3
    );
END_TYPE

// ---- Library/10_Machine/18_HMI_Handshake/DUTs/Allocated/ST_Auto_Allocated.TcDUT
TYPE
    ST_Auto_Allocated :
    STRUCT
    END_STRUCT
END_TYPE

// ---- Library/10_Machine/18_HMI_Handshake/DUTs/Allocated/ST_AXIS_HOMING.TcDUT
TYPE ST_AXIS_HOMING :
    STRUCT
        Execute : BOOL; // True : start homing process
        Abort   : BOOL; // True : abort homing process
    END_STRUCT
END_TYPE

// ---- Library/10_Machine/18_HMI_Handshake/DUTs/Allocated/ST_AXIS_JOG.TcDUT
TYPE ST_AXIS_JOG :
STRUCT
	MoveFWD : BOOL; // Axis Jog control, move forward
	MoveBWD : BOOL; // Axis Jog control, move backward
END_STRUCT
END_TYPE

// ---- Library/10_Machine/18_HMI_Handshake/DUTs/Allocated/ST_AXIS_PTP.TcDUT
TYPE
    ST_AXIS_PTP :
    STRUCT
		Enable 		 : BOOL; // True : Position Absolute mode active
        Position     : LREAL; // The position command during PTP (Point-to-Point) positioning.
        Velocity     : LREAL; // The velocity command during PTP (Point-to-Point) positioning.
        Acceleration : LREAL; // The acceleration command during PTP (Point-to-Point) positioning.
        Deceleration : LREAL; // The deceleration command during PTP (Point-to-Point) positioning.
        Jerk         : LREAL; // The jerk command during PTP (Point-to-Point) positioning.
    END_STRUCT
END_TYPE

// ---- Library/10_Machine/18_HMI_Handshake/DUTs/Allocated/ST_HalfAuto_Allocated.TcDUT
TYPE
    ST_HalfAuto_Allocated :
    STRUCT
        TableMove : ST_TableMoveService; // When machine in Manual mode, it can trig execute to move module to targer position with PositionTable
    END_STRUCT
END_TYPE

// ---- Library/10_Machine/18_HMI_Handshake/DUTs/Allocated/ST_HMI_ControlOutPut.TcDUT
TYPE
    ST_HMI_ControlOutPut :
    STRUCT      
		FanucRobot	    : ST_Manual_FanucRobot; 	//六軸手臂行動命令
		RackMotor 	    : ST_Manual_Axis;			//補貨料架馬達行動命令
		OutRobot        : ST_Manual_OutRobot;       //出料手臂行動命令
        NeedleRobot     : ST_Manual_NeedleRobot; 	//配針手臂行動命令
        Allocate        : ST_Manual_Allocate;     	//圓帶行動命令
        TurnTable       : ST_Manual_TurnTable;      //圓盤行動命令 
		ElvaterAxis		: ST_Manual_Axis;			//電梯行動命令
		HookAxis		: ST_Manual_Axis;			//勾盤行動命令
		FinishAxis		: ST_Manual_Axis;			//出料層架行動命令
 END_STRUCT
END_TYPE

// ---- Library/10_Machine/18_HMI_Handshake/DUTs/Allocated/ST_Manual_Allocated.TcDUT
TYPE
    ST_Manual_Allocated :
    STRUCT
        OutRobot       : ST_Manual_OutRobot;       // Allocated out robot manual control
        NeedleRobot    : ST_Manual_NeedleRobot; // Allocated allocated robot manual control
        Allocate       : ST_Manual_Allocate;      // Allocated round belt manual control
        TurnTable      : ST_Manual_TurnTable;      // Allocated turn table manual control
        PullOutCV      : ST_Manual_PullOutCV;        // Allocated pullout conveyor manual control
        TransCV        : ST_Manual_TransCV;        // Allocated transmit conveyor manual control
    END_STRUCT
END_TYPE

// ---- Library/10_Machine/18_HMI_Handshake/DUTs/Allocated/ST_Manual_NeedleRobot.TcDUT
TYPE
    ST_Manual_NeedleRobot :
    STRUCT
        LeftVert1   : ST_SignleValve; // AllocateRobot LeftVert1 cylinder controll
        LeftVert2   : ST_SignleValve; // AllocateRobot LeftVert2 cylinder controll
        RightVert1  : ST_SignleValve; // AllocateRobot RightVert1 cylinder controll
        RightVert2  : ST_SignleValve; // AllocateRobot RightVert2 cylinder controll
        LeftClamp1  : ST_SignleValve; // AllocateRobot LeftClamp1 cylinder controll
        LeftClamp2  : ST_SignleValve; // AllocateRobot LeftClamp2 cylinder controll
        RightClamp1 : ST_SignleValve; // AllocateRobot RightClamp1 cylinder controll
        RightClamp2 : ST_SignleValve; // AllocateRobot RightClamp2 cylinder controll
        AxisX       : ST_Manual_Axis; // AllocateRobot AxisX controll
        AxisY       : ST_Manual_Axis; // AllocateRobot AxisY controll
    END_STRUCT
END_TYPE

// ---- Library/10_Machine/18_HMI_Handshake/DUTs/Allocated/ST_Manual_Axis.TcDUT
TYPE ST_Manual_Axis :
STRUCT
	JOGMoveFWD 		: BOOL; // Axis Jog control, move forward
	JOGMoveBWD 		: BOOL; // Axis Jog control, move backward
	PTPEnable 		: BOOL; // True : Position Absolute mode active
    PTPPosition     : LREAL; // The position command during PTP (Point-to-Point) positioning.
    PTPVelocity     : LREAL; // The velocity command during PTP (Point-to-Point) positioning.
    PTPAcceleration : LREAL; // The acceleration command during PTP (Point-to-Point) positioning.
    PTPDeceleration : LREAL; // The deceleration command during PTP (Point-to-Point) positioning.
    PTPJerk         : LREAL; // The jerk command during PTP (Point-to-Point) positioning.
	Homing 			: ST_AXIS_HOMING;
END_STRUCT
END_TYPE

// ---- Library/10_Machine/18_HMI_Handshake/DUTs/Allocated/ST_Manual_OutRobot.TcDUT
TYPE
    ST_Manual_OutRobot :
    STRUCT
        AsideVert  : ST_SignleValve; // OutRobot AsideVert cylinder controll
        BsideVert  : ST_SignleValve; // OutRobot BsideVert cylinder controll
        AsideClamp : ST_SignleValve; // OutRobot AsideClamp cylinder controll
        BsideClamp : ST_SignleValve; // OutRobot BsideClamp cylinder controll
        AxisX      : ST_Manual_Axis; // OutRobot AxisX controll
        AxisY      : ST_Manual_Axis; // OutRobot AxisY controll
    END_STRUCT
END_TYPE

// ---- Library/10_Machine/18_HMI_Handshake/DUTs/Allocated/ST_Manual_PullOutCV.TcDUT
TYPE
    ST_Manual_PullOutCV :
    STRUCT
        AsidePress1 : ST_SignleValve;
        AsidePress2 : ST_SignleValve;
        AsideBlock  : ST_SignleValve;
        BsidePress1 : ST_SignleValve;
        BsidePress2 : ST_SignleValve;
        BsideBlock  : ST_SignleValve;
        PullOutCV_A : ST_MotorCommand;
        PullOutCV_B : ST_MotorCommand;
    END_STRUCT
END_TYPE

// ---- Library/10_Machine/18_HMI_Handshake/DUTs/Allocated/ST_Manual_Allocate.TcDUT
TYPE
    ST_Manual_Allocate :
    STRUCT
        WorkZone_Press      : ST_SignleValve;
        WorkZone_Plug       : ST_SignleValve; //定位銷
        ChargeZone_Plug     : ST_SignleValve; //定位銷
        TransmitCVZone_Plug : ST_SignleValve; //定位銷
        Axis                : ST_Manual_Axis; // RoundBelt Axis controll
		
    END_STRUCT
END_TYPE

// ---- Library/10_Machine/18_HMI_Handshake/DUTs/Allocated/ST_Manual_TransCV.TcDUT
TYPE
    ST_Manual_TransCV :
    STRUCT
        DifferentSizeCV_Press2  : ST_SignleValve;
        DifferentSizeCV_Press1  : ST_SignleValve;
        DifferentSizeCV_Block1  : ST_SignleValve;
        SameSizeCV_Press4       : ST_SignleValve;
        SameSizeCV_Press3       : ST_SignleValve;
        SameSizeCV_Press2       : ST_SignleValve;
        SameSizeCV_Press1       : ST_SignleValve;
        SameSizeCV_Block2       : ST_SignleValve;
        SameSizeCV_Block1       : ST_SignleValve;
        TransmitSameSideCV      : ST_MotorCommand;
        TransmitDifferentSideCV : ST_MotorCommand;
    END_STRUCT
END_TYPE

// ---- Library/10_Machine/18_HMI_Handshake/DUTs/Allocated/ST_Manual_TurnTable.TcDUT
TYPE
    ST_Manual_TurnTable :
    STRUCT
        Press : ST_SignleValve;
        Axis  : ST_Manual_Axis; // TurnTable Axis controll
    END_STRUCT
END_TYPE

// ---- Library/10_Machine/18_HMI_Handshake/DUTs/Component/ST_DoubleValve.TcDUT
TYPE
    ST_DoubleValve EXTENDS ST_SignleValve :
    STRUCT
        Retract : BOOL;
    END_STRUCT
END_TYPE

// ---- Library/10_Machine/18_HMI_Handshake/DUTs/Component/ST_MotorCommand.TcDUT
TYPE
    ST_MotorCommand :
    STRUCT
        Forward  : BOOL;
        Backward : BOOL;
        Stopped  : BOOL;
    END_STRUCT
END_TYPE

// ---- Library/10_Machine/18_HMI_Handshake/DUTs/Component/ST_SignleValve.TcDUT
TYPE
    ST_SignleValve :
    STRUCT
        Exetend : BOOL;
    END_STRUCT
END_TYPE

// ---- Library/10_Machine/18_HMI_Handshake/DUTs/E_AllocationJob.TcDUT
{attribute 'qualified_only'}
{attribute 'strict'}
TYPE E_AllocationJob :
(	PreDataProcess:=-1,
	Idle:=0,	
	Initial ,	
	CheckRotateBeltStation,
	MovingRotateBeltStation,
	MovedRotateBeltStation,
	CheckRotateBeltStation_SimpleAllocatePlacing,
	MovingRotateBeltStation_SimpleAllocatePlacing,
	MovedRotateBeltStation_SimpleAllocatePlacing,
	CheckBoxReadyOnAllocatePosOfRoundBelt,
	CheckBoxReadyOnRoundBelt_SimpleAllocateMode,
	MoveToTargetPos,
	MovingToTargetPos,
	CylinderDownPick,
	ClipColse,	
	CylinderUpPick,
	MoveToPlacingPos,
	MovingToPlacingPos,
	CylinderDownPlace,
	ClipOpen,		
	CylinderUpPlace,
	CheckNeedlePlaced,
	Defult,
	Finish,
	Error,
	CheckNeedlePick,
	CheckNeedlePlace,
	IfNextPTP_Picking,
	IfNextPTP_Placing,
	CheckBoxesOnTurnTableReady	
	
);
END_TYPE

// ---- Library/10_Machine/18_HMI_Handshake/DUTs/IOMonitor/ST_HMI_ControlInPut.TcDUT
TYPE
    ST_HMI_ControlInPut :
    STRUCT
        Input  : ST_InputTables;
        Output : ST_OutputTables;
    END_STRUCT
END_TYPE

// ---- Library/10_Machine/18_HMI_Handshake/DUTs/IOMonitor/ST_InputTables.TcDUT
TYPE ST_InputTables :
STRUCT
	    X6  : uni_IntToBool;
        X7  : uni_IntToBool;
        X9  : uni_IntToBool;
        X10 : uni_IntToBool;
        X0  : uni_IntToBool;
        X1  : uni_IntToBool;
        X2  : uni_IntToBool;
        X3  : uni_IntToBool;
        X8  : uni_IntToBool;
        X11 : uni_IntToBool;
        X4  : uni_IntToBool;
		arWheelhouseInput : ARRAY[1..400] OF BOOL;
END_STRUCT
END_TYPE

// ---- Library/10_Machine/18_HMI_Handshake/DUTs/IOMonitor/ST_Input_IOMonitor.TcDUT
TYPE
    ST_Input_IOMonitor :
    STRUCT
    END_STRUCT
END_TYPE

// ---- Library/10_Machine/18_HMI_Handshake/DUTs/IOMonitor/ST_Output_IOMonitor.TcDUT
TYPE
    ST_Output_IOMonitor :
    STRUCT
    END_STRUCT
END_TYPE

// ---- Library/10_Machine/18_HMI_Handshake/DUTs/IOMonitor/ST_WheelhouseInput.TcDUT
TYPE
    ST_WheelhouseInput :
    STRUCT
        WheelhouseA : ST_WheelhouseTour;
        WheelhouseB : ST_WheelhouseTour;
    END_STRUCT
END_TYPE

// ---- Library/10_Machine/18_HMI_Handshake/DUTs/IOMonitor/ST_WheelhouseTour.TcDUT
TYPE
    ST_WheelhouseTour :
    STRUCT
        arLayer : ARRAY[1..10] OF ST_Wheelhouse_Layer;
    END_STRUCT
END_TYPE

